C01876=52.817,75.362,62.469,-177.2451,7.5721,0.0000
C01877=50.052,70.729,61.698,-175.7549,6.7538,0.0000
C01878=46.818,66.007,60.151,-176.6982,5.1590,0.0000
C01879=43.998,61.798,58.158,-178.4123,2.6620,0.0000
C01880=42.158,58.431,56.252,178.4711,-3.3109,0.0000
C01881=41.963,55.679,54.888,-171.7704,-29.0710,0.0000
C01882=44.137,52.905,54.350,-151.3798,-29.7512,0.0000
C01883=46.553,50.718,54.326,-149.2273,-28.3546,0.0000
C01884=48.679,48.679,54.342,-150.4011,-29.5986,0.0000
C01885=50.718,46.553,54.326,-151.6456,-30.7729,0.0000
C01886=52.905,44.137,54.350,-150.2477,-28.6184,0.0000
C01887=55.680,41.963,54.888,-150.9289,-8.2300,0.0000
C01888=58.431,42.158,56.252,-176.6891,1.5289,0.0000
C01889=61.798,43.998,58.158,177.3380,-1.5877,0.0000
C01890=66.007,46.818,60.151,174.8410,-3.3018,0.0000
C01891=70.729,50.052,61.698,173.2462,-4.2451,0.0000
C01892=75.362,52.817,62.469,172.4279,-2.7549,0.0000
C01893=80.376,53.158,62.877,175.1551,1.0270,0.0000
C01894=85.074,50.908,63.210,178.0786,1.5643,0.0000
C01895=88.493,46.465,63.547,179.9251,0.1391,0.0000
C01896=91.166,41.080,63.770,179.9921,0.0174,0.0000
C01897=93.512,35.416,63.770,179.9933,0.0179,0.0000
C01898=95.429,29.718,63.547,179.9546,0.1514,0.0000
C01899=96.154,24.159,63.210,-179.7472,2.4641,0.0000
C01900=94.423,19.246,62.877,-177.2942,4.1530,0.0000
C01901=90.636,15.942,62.469,-172.7045,3.4321,0.0000
C01902=85.405,14.621,61.698,-172.2425,1.7901,0.0000
C01903=79.780,13.569,60.151,-174.0266,1.3203,0.0000
C01904=74.809,12.586,58.158,-176.9961,0.7607,0.0000
C01905=71.127,11.507,56.252,176.5790,-1.2623,0.0000
C01906=69.044,9.699,54.888,163.7838,-26.3525,0.0000
C01907=68.619,6.200,54.350,178.9508,-38.3093,0.0000
C01908=68.781,2.945,54.326,-177.7405,-38.7530,0.0000
C01909=68.843,0.000,54.342,-179.9996,-38.7765,0.0000
C01910=68.781,-2.945,54.326,177.7401,-38.7530,0.0000
C01911=68.619,-6.200,54.350,-178.9482,-38.3089,0.0000
C01912=69.044,-9.699,54.888,-163.7840,-26.3528,0.0000
C01913=71.127,-11.507,56.252,-176.5790,-1.2623,0.0000
C01914=74.809,-12.586,58.158,176.9961,0.7607,0.0000
C01915=79.780,-13.569,60.151,174.0266,1.3203,0.0000
C01916=85.405,-14.621,61.698,172.2425,1.7901,0.0000
C01917=90.636,-15.942,62.469,172.7045,3.4321,0.0000
C01918=94.423,-19.246,62.877,177.2942,4.1530,0.0000
C01919=96.154,-24.159,63.210,179.7472,2.4641,0.0000
C01920=95.429,-29.718,63.547,-179.9546,0.1514,0.0000
C01921=93.512,-35.416,63.770,-179.9933,0.0179,0.0000
C01922=91.166,-41.080,63.770,-179.9921,0.0174,0.0000
C01923=88.493,-46.465,63.547,-179.9251,0.1391,0.0000
C01924=85.074,-50.908,63.210,-178.0786,1.5643,0.0000
C01925=80.376,-53.158,62.877,-175.1551,1.0270,0.0000
C01926=75.362,-52.817,62.469,-172.4279,-2.7549,0.0000
C01927=70.729,-50.052,61.698,-173.2462,-4.2451,0.0000
C01928=66.007,-46.818,60.151,-174.8410,-3.3018,0.0000
C01929=61.798,-43.998,58.158,-177.3380,-1.5877,0.0000
C01930=58.431,-42.158,56.252,176.6891,1.5289,0.0000
C01931=55.679,-41.963,54.888,150.9290,-8.2296,0.0000
C01932=52.905,-44.137,54.350,150.2488,-28.6202,0.0000
C01933=50.718,-46.553,54.326,151.6454,-30.7727,0.0000
C01934=48.679,-48.679,54.342,150.4014,-29.5989,0.0000
C01935=46.553,-50.718,54.326,149.2271,-28.3544,0.0000
C01936=44.137,-52.905,54.350,151.3816,-29.7523,0.0000
C01937=41.963,-55.680,54.888,171.7700,-29.0711,0.0000
C01938=42.158,-58.431,56.252,-178.4711,-3.3109,0.0000
C01939=43.998,-61.798,58.158,178.4123,2.6620,0.0000
C01940=46.818,-66.007,60.151,176.6982,5.1590,0.0000
C01941=50.052,-70.729,61.698,175.7549,6.7538,0.0000
C01942=52.817,-75.362,62.469,177.2451,7.5721,0.0000
C01943=53.158,-80.376,62.877,-178.9730,4.8449,0.0000
C01944=50.908,-85.074,63.210,-178.4357,1.9214,0.0000
C01945=46.465,-88.493,63.547,-179.8609,0.0749,0.0000
C01946=41.080,-91.166,63.770,-179.9826,0.0079,0.0000
C01947=35.416,-93.512,63.770,-179.9821,0.0067,0.0000
C01948=29.718,-95.429,63.547,-179.8486,0.0454,0.0000
C01949=24.159,-96.154,63.210,-177.5359,-0.2528,0.0000
C01950=19.246,-94.423,62.877,-175.8470,-2.7058,0.0000
C01951=15.942,-90.636,62.469,-176.5679,-7.2955,0.0000
C01952=14.621,-85.405,61.698,-178.2099,-7.7575,0.0000
C01953=13.569,-79.780,60.151,-178.6797,-5.9734,0.0000
C01954=12.586,-74.809,58.158,-179.2393,-3.0039,0.0000
C01955=11.507,-71.127,56.252,178.7377,3.4210,0.0000
C01956=9.699,-69.044,54.888,153.6475,16.2162,0.0000
C01957=6.200,-68.619,54.350,141.6907,1.0492,0.0000
C01958=2.945,-68.781,54.326,141.2470,-2.2595,0.0000
C01959=0.000,-68.843,54.342,141.2235,-0.0004,0.0000
C01960=0.000,-68.843,54.342,141.2235,-0.0004,0.0000
C01961=-2.945,-68.781,54.326,141.2470,2.2599,0.0000
C01962=-6.200,-68.619,54.350,141.6911,-1.0518,0.0000
C01963=-9.699,-69.044,54.888,153.6472,-16.2160,0.0000
C01964=-11.507,-71.127,56.252,178.7377,-3.4210,0.0000
C01965=-12.586,-74.809,58.158,-179.2393,3.0039,0.0000
C01966=-13.569,-79.780,60.151,-178.6797,5.9734,0.0000
C01967=-14.621,-85.405,61.698,-178.2099,7.7575,0.0000
C01968=-15.942,-90.636,62.469,-176.5679,7.2955,0.0000
C01969=-19.246,-94.423,62.877,-175.8470,2.7058,0.0000
C01970=-24.159,-96.154,63.210,-177.5359,0.2528,0.0000
C01971=-29.718,-95.429,63.547,-179.8486,-0.0454,0.0000
C01972=-35.416,-93.512,63.770,-179.9821,-0.0067,0.0000
C01973=-41.080,-91.166,63.770,-179.9826,-0.0079,0.0000
C01974=-46.465,-88.493,63.547,-179.8609,-0.0749,0.0000
C01975=-50.908,-85.074,63.210,-178.4357,-1.9214,0.0000
C01976=-53.158,-80.376,62.877,-178.9730,-4.8449,0.0000
C01977=-52.817,-75.362,62.469,177.2451,-7.5721,0.0000
C01978=-50.052,-70.729,61.698,175.7549,-6.7538,0.0000
C01979=-46.818,-66.007,60.151,176.6982,-5.1590,0.0000
C01980=-43.998,-61.798,58.158,178.4123,-2.6620,0.0000
C01981=-42.158,-58.431,56.252,-178.4711,3.3109,0.0000
C01982=-41.963,-55.679,54.888,171.7704,29.0710,0.0000
C01983=-44.137,-52.905,54.350,151.3798,29.7512,0.0000
C01984=-46.553,-50.718,54.326,149.2273,28.3546,0.0000
C01985=-48.679,-48.679,54.342,150.4011,29.5986,0.0000
C01986=-50.718,-46.553,54.326,151.6456,30.7729,0.0000
C01987=-52.905,-44.137,54.350,150.2477,28.6184,0.0000
C01988=-55.680,-41.963,54.888,150.9289,8.2300,0.0000
C01989=-58.431,-42.158,56.252,176.6891,-1.5289,0.0000
C01990=-61.798,-43.998,58.158,-177.3380,1.5877,0.0000
C01991=-66.007,-46.818,60.151,-174.8410,3.3018,0.0000
C01992=-70.729,-50.052,61.698,-173.2462,4.2451,0.0000
C01993=-75.362,-52.817,62.469,-172.4279,2.7549,0.0000
C01994=-80.376,-53.158,62.877,-175.1551,-1.0270,0.0000
C01995=-85.074,-50.908,63.210,-178.0786,-1.5643,0.0000
C01996=-88.493,-46.465,63.547,-179.9251,-0.1391,0.0000
C01997=-91.166,-41.080,63.770,-179.9921,-0.0174,0.0000
C01998=-93.512,-35.416,63.770,-179.9933,-0.0179,0.0000
C01999=-95.429,-29.718,63.547,-179.9546,-0.1514,0.0000
///TOOL 0
///POSTYPE ANGLE
///ANGLE
EC00000=-73.7963,0.0000
EC00001=-71.3299,0.0000
EC00002=-68.7820,0.0000
EC00003=-66.2179,0.0000
EC00004=-63.6703,0.0000
EC00005=-61.2039,0.0000
EC00006=-59.0550,0.0000
EC00007=-57.5413,0.0000
EC00008=-56.8513,0.0000
EC00009=-56.3680,0.0000
EC00010=-55.8386,0.0000
EC00011=-55.0278,0.0000
EC00012=-53.5081,0.0000
EC00013=-50.7770,0.0000
EC00014=-47.9180,0.0000
EC00015=-45.0000,0.0000
EC00016=-42.0820,0.0000
EC00017=-39.2230,0.0000
EC00018=-36.4919,0.0000
EC00019=-34.9722,0.0000
EC00020=-34.1614,0.0000
EC00021=-33.6320,0.0000
EC00022=-33.1487,0.0000
EC00023=-32.4587,0.0000
EC00024=-30.9450,0.0000
EC00025=-28.7961,0.0000
EC00026=-26.3297,0.0000
EC00027=-23.7821,0.0000
EC00028=-21.2180,0.0000
EC00029=-18.6701,0.0000
EC00030=-16.2037,0.0000
EC00031=-14.0550,0.0000
EC00032=-12.5410,0.0000
EC00033=-11.8512,0.0000
EC00034=-11.3683,0.0000
EC00035=-10.8382,0.0000
EC00036=-10.0280,0.0000
EC00037=-8.5076,0.0000
EC00038=-5.7775,0.0000
EC00039=-2.9180,0.0000
EC00040=0.0000,0.0000
EC00041=0.0000,0.0000
EC00042=2.8792,0.0000
EC00043=5.7259,0.0000
EC00044=8.4654,0.0000
EC00045=9.9566,0.0000
EC00046=10.7254,0.0000
EC00047=11.2119,0.0000
EC00048=11.6495,0.0000
EC00049=12.2909,0.0000
EC00050=13.8024,0.0000
EC00051=15.9922,0.0000
EC00052=18.5312,0.0000
EC00053=21.1696,0.0000
EC00054=23.8303,0.0000
EC00055=26.4689,0.0000
EC00056=29.0082,0.0000
EC00057=31.1977,0.0000
EC00058=32.7089,0.0000
EC00059=33.3509,0.0000
EC00060=33.7878,0.0000
EC00061=34.2746,0.0000
EC00062=35.0436,0.0000
EC00063=36.5348,0.0000
EC00064=39.2737,0.0000
EC00065=42.1206,0.0000
EC00066=45.0000,0.0000
EC00067=47.8789,0.0000
EC00068=50.7263,0.0000
EC00069=53.4652,0.0000
EC00070=54.9564,0.0000
EC00071=55.7254,0.0000
EC00072=56.2122,0.0000
EC00073=56.6491,0.0000
EC00074=57.2911,0.0000
EC00075=58.8023,0.0000
EC00076=60.9918,0.0000
EC00077=63.5311,0.0000
EC00078=66.1697,0.0000
EC00079=68.8304,0.0000
EC00080=71.4688,0.0000
EC00081=74.0078,0.0000
EC00082=76.1976,0.0000
EC00083=77.7091,0.0000
EC00084=78.3505,0.0000
EC00085=78.7881,0.0000
EC00086=79.2746,0.0000
EC00087=80.0434,0.0000
EC00088=81.5346,0.0000
EC00089=84.2741,0.0000
EC00090=87.1208,0.0000
EC00091=90.0000,0.0000
EC00092=92.8792,0.0000
EC00093=95.7266,0.0000
EC00094=98.4654,0.0000
EC00095=99.9566,0.0000
EC00096=100.7254,0.0000
EC00097=101.2119,0.0000
EC00098=101.6495,0.0000
EC00099=102.2909,0.0000
EC00100=103.8024,0.0000
EC00101=105.9922,0.0000
EC00102=108.5312,0.0000
EC00103=111.1696,0.0000
EC00104=113.8303,0.0000
EC00105=116.4689,0.0000
EC00106=119.0082,0.0000
EC00107=121.1977,0.0000
EC00108=122.7089,0.0000
EC00109=123.3509,0.0000
EC00110=123.7878,0.0000
EC00111=124.2746,0.0000
EC00112=125.0436,0.0000
EC00113=126.5348,0.0000
EC00114=129.2737,0.0000
EC00115=132.1206,0.0000
EC00116=135.0000,0.0000
EC00117=137.8789,0.0000
EC00118=140.7263,0.0000
EC00119=143.4652,0.0000
EC00120=144.9564,0.0000
EC00121=145.7254,0.0000
EC00122=146.2122,0.0000
EC00123=146.6491,0.0000
EC00124=147.2911,0.0000
EC00125=148.8023,0.0000
EC00126=150.9918,0.0000
EC00127=153.5311,0.0000
EC00128=156.1697,0.0000
EC00129=158.8304,0.0000
EC00130=161.4688,0.0000
EC00131=164.0078,0.0000
EC00132=166.1976,0.0000
EC00133=167.7091,0.0000
EC00134=168.3505,0.0000
EC00135=168.7881,0.0000
EC00136=169.2746,0.0000
EC00137=170.0434,0.0000
EC00138=171.5346,0.0000
EC00139=174.2741,0.0000
EC00140=177.1208,0.0000
EC00141=180.0000,0.0000
EC00142=180.0000,0.0000
EC00143=-177.1208,0.0000
EC00144=-174.2734,0.0000
EC00145=-171.5346,0.0000
EC00146=-170.0434,0.0000
EC00147=-169.2746,0.0000
EC00148=-168.7881,0.0000
EC00149=-168.3505,0.0000
EC00150=-167.7091,0.0000
EC00151=-166.1976,0.0000
EC00152=-164.0078,0.0000
EC00153=-161.4688,0.0000
EC00154=-158.8304,0.0000
EC00155=-156.1697,0.0000
EC00156=-153.5311,0.0000
EC00157=-150.9918,0.0000
EC00158=-148.8023,0.0000
EC00159=-147.2911,0.0000
EC00160=-146.6491,0.0000
EC00161=-146.2122,0.0000
EC00162=-145.7254,0.0000
EC00163=-144.9564,0.0000
EC00164=-143.4652,0.0000
EC00165=-140.7263,0.0000
EC00166=-137.8794,0.0000
EC00167=-135.0000,0.0000
EC00168=-132.1211,0.0000
EC00169=-129.2737,0.0000
EC00170=-126.5348,0.0000
EC00171=-125.0436,0.0000
EC00172=-124.2746,0.0000
EC00173=-123.7878,0.0000
EC00174=-123.3509,0.0000
EC00175=-122.7089,0.0000
EC00176=-121.1977,0.0000
EC00177=-119.0082,0.0000
EC00178=-116.4689,0.0000
EC00179=-113.8303,0.0000
EC00180=-111.1696,0.0000
EC00181=-108.5312,0.0000
EC00182=-105.9922,0.0000
EC00183=-103.8024,0.0000
EC00184=-102.2909,0.0000
EC00185=-101.6495,0.0000
EC00186=-101.2119,0.0000
EC00187=-100.7254,0.0000
EC00188=-99.9566,0.0000
EC00189=-98.4654,0.0000
EC00190=-95.7259,0.0000
EC00191=-92.8792,0.0000
EC00192=-90.0000,0.0000
EC00193=-87.1208,0.0000
EC00194=-84.2734,0.0000
EC00195=-81.5346,0.0000
EC00196=-80.0434,0.0000
EC00197=-79.2746,0.0000
EC00198=-78.7881,0.0000
EC00199=-78.3505,0.0000
EC00200=-77.7091,0.0000
EC00201=-76.1976,0.0000
EC00202=-74.0078,0.0000
EC00203=-71.4688,0.0000
EC00204=-68.8304,0.0000
EC00205=-66.1697,0.0000
EC00206=-63.5311,0.0000
EC00207=-60.9918,0.0000
EC00208=-58.8023,0.0000
EC00209=-57.2911,0.0000
EC00210=-56.6491,0.0000
EC00211=-56.2122,0.0000
EC00212=-55.7254,0.0000
EC00213=-54.9564,0.0000
EC00214=-53.4652,0.0000
EC00215=-50.7263,0.0000
EC00216=-47.8794,0.0000
EC00217=-45.0000,0.0000
EC00218=-42.1211,0.0000
EC00219=-39.2737,0.0000
EC00220=-36.5348,0.0000
EC00221=-35.0436,0.0000
EC00222=-34.2746,0.0000
EC00223=-33.7878,0.0000
EC00224=-33.3509,0.0000
EC00225=-32.7089,0.0000
EC00226=-31.1977,0.0000
EC00227=-29.0082,0.0000
EC00228=-26.4689,0.0000
EC00229=-23.8303,0.0000
EC00230=-21.1696,0.0000
EC00231=-18.5312,0.0000
EC00232=-15.9922,0.0000
EC00233=-13.8024,0.0000
EC00234=-12.2909,0.0000
EC00235=-11.6495,0.0000
EC00236=-11.2119,0.0000
EC00237=-10.7254,0.0000
EC00238=-9.9566,0.0000
EC00239=-8.4654,0.0000
EC00240=-5.7266,0.0000
EC00241=-2.8792,0.0000
EC00242=0.0000,0.0000
EC00243=0.0000,0.0000
EC00244=2.8388,0.0000
EC00245=5.6728,0.0000
EC00246=8.4202,0.0000
EC00247=9.8823,0.0000
EC00248=10.6084,0.0000
EC00249=11.0516,0.0000
EC00250=11.4429,0.0000
EC00251=12.0370,0.0000
EC00252=13.5473,0.0000
EC00253=15.7781,0.0000
EC00254=18.3907,0.0000
EC00255=21.1209,0.0000
EC00256=23.8793,0.0000
EC00257=26.6097,0.0000
EC00258=29.2218,0.0000
EC00259=31.4529,0.0000
EC00260=32.9628,0.0000
EC00261=33.5569,0.0000
EC00262=33.9481,0.0000
EC00263=34.3909,0.0000
EC00264=35.1173,0.0000
EC00265=36.5793,0.0000
EC00266=39.3269,0.0000
EC00267=42.1606,0.0000
EC00268=45.0000,0.0000
EC00269=47.8388,0.0000
EC00270=50.6731,0.0000
EC00271=53.4207,0.0000
EC00272=54.8827,0.0000
EC00273=55.6091,0.0000
EC00274=56.0519,0.0000
EC00275=56.4431,0.0000
EC00276=57.0372,0.0000
EC00277=58.5471,0.0000
EC00278=60.7782,0.0000
EC00279=63.3903,0.0000
EC00280=66.1207,0.0000
EC00281=68.8791,0.0000
EC00282=71.6093,0.0000
EC00283=74.2219,0.0000
EC00284=76.4527,0.0000
EC00285=77.9630,0.0000
EC00286=78.5571,0.0000
EC00287=78.9484,0.0000
EC00288=79.3916,0.0000
EC00289=80.1177,0.0000
EC00290=81.5798,0.0000
EC00291=84.3272,0.0000
EC00292=87.1612,0.0000
EC00293=90.0000,0.0000
EC00294=92.8388,0.0000
EC00295=95.6728,0.0000
EC00296=98.4209,0.0000
EC00297=99.8823,0.0000
EC00298=100.6084,0.0000
EC00299=101.0516,0.0000
EC00300=101.4429,0.0000
EC00301=102.0370,0.0000
EC00302=103.5473,0.0000
EC00303=105.7781,0.0000
EC00304=108.3907,0.0000
EC00305=111.1209,0.0000
EC00306=113.8793,0.0000
EC00307=116.6097,0.0000
EC00308=119.2218,0.0000
EC00309=121.4529,0.0000
EC00310=122.9628,0.0000
EC00311=123.5569,0.0000
EC00312=123.9481,0.0000
EC00313=124.3909,0.0000
EC00314=125.1173,0.0000
EC00315=126.5793,0.0000
EC00316=129.3269,0.0000
EC00317=132.1606,0.0000
EC00318=135.0000,0.0000
EC00319=137.8388,0.0000
EC00320=140.6731,0.0000
EC00321=143.4207,0.0000
EC00322=144.8827,0.0000
EC00323=145.6091,0.0000
EC00324=146.0519,0.0000
EC00325=146.4431,0.0000
EC00326=147.0372,0.0000
EC00327=148.5471,0.0000
EC00328=150.7782,0.0000
EC00329=153.3903,0.0000
EC00330=156.1207,0.0000
EC00331=158.8791,0.0000
EC00332=161.6093,0.0000
EC00333=164.2219,0.0000
EC00334=166.4527,0.0000
EC00335=167.9630,0.0000
EC00336=168.5571,0.0000
EC00337=168.9484,0.0000
EC00338=169.3916,0.0000
EC00339=170.1177,0.0000
EC00340=171.5798,0.0000
EC00341=174.3272,0.0000
EC00342=177.1612,0.0000
EC00343=180.0000,0.0000
EC00344=180.0000,0.0000
EC00345=-177.1612,0.0000
EC00346=-174.3272,0.0000
EC00347=-171.5791,0.0000
EC00348=-170.1177,0.0000
EC00349=-169.3916,0.0000
EC00350=-168.9484,0.0000
EC00351=-168.5571,0.0000
EC00352=-167.9630,0.0000
EC00353=-166.4527,0.0000
EC00354=-164.2219,0.0000
EC00355=-161.6093,0.0000
EC00356=-158.8791,0.0000
EC00357=-156.1207,0.0000
EC00358=-153.3903,0.0000
EC00359=-150.7782,0.0000
EC00360=-148.5471,0.0000
EC00361=-147.0372,0.0000
EC00362=-146.4431,0.0000
EC00363=-146.0519,0.0000
EC00364=-145.6091,0.0000
EC00365=-144.8827,0.0000
EC00366=-143.4207,0.0000
EC00367=-140.6731,0.0000
EC00368=-137.8394,0.0000
EC00369=-135.0000,0.0000
EC00370=-132.1612,0.0000
EC00371=-129.3269,0.0000
EC00372=-126.5793,0.0000
EC00373=-125.1173,0.0000
EC00374=-124.3909,0.0000
EC00375=-123.9481,0.0000
EC00376=-123.5569,0.0000
EC00377=-122.9628,0.0000
EC00378=-121.4529,0.0000
EC00379=-119.2218,0.0000
EC00380=-116.6097,0.0000
EC00381=-113.8793,0.0000
EC00382=-111.1209,0.0000
EC00383=-108.3907,0.0000
EC00384=-105.7781,0.0000
EC00385=-103.5473,0.0000
EC00386=-102.0370,0.0000
EC00387=-101.4429,0.0000
EC00388=-101.0516,0.0000
EC00389=-100.6084,0.0000
EC00390=-99.8823,0.0000
EC00391=-98.4202,0.0000
EC00392=-95.6728,0.0000
EC00393=-92.8388,0.0000
EC00394=-90.0000,0.0000
EC00395=-87.1612,0.0000
EC00396=-84.3272,0.0000
EC00397=-81.5791,0.0000
EC00398=-80.1177,0.0000
EC00399=-79.3916,0.0000
EC00400=-78.9484,0.0000
EC00401=-78.5571,0.0000
EC00402=-77.9630,0.0000
EC00403=-76.4527,0.0000
EC00404=-74.2219,0.0000
EC00405=-71.6093,0.0000
EC00406=-68.8791,0.0000
EC00407=-66.1207,0.0000
EC00408=-63.3903,0.0000
EC00409=-60.7782,0.0000
EC00410=-58.5471,0.0000
EC00411=-57.0372,0.0000
EC00412=-56.4431,0.0000
EC00413=-56.0519,0.0000
EC00414=-55.6091,0.0000
EC00415=-54.8827,0.0000
EC00416=-53.4207,0.0000
EC00417=-50.6731,0.0000
EC00418=-47.8394,0.0000
EC00419=-45.0000,0.0000
EC00420=-42.1612,0.0000
EC00421=-39.3269,0.0000
EC00422=-36.5793,0.0000
EC00423=-35.1173,0.0000
EC00424=-34.3909,0.0000
EC00425=-33.9481,0.0000
EC00426=-33.5569,0.0000
EC00427=-32.9628,0.0000
EC00428=-31.4529,0.0000
EC00429=-29.2218,0.0000
EC00430=-26.6097,0.0000
EC00431=-23.8793,0.0000
EC00432=-21.1209,0.0000
EC00433=-18.3907,0.0000
EC00434=-15.7781,0.0000
EC00435=-13.5473,0.0000
EC00436=-12.0370,0.0000
EC00437=-11.4429,0.0000
EC00438=-11.0516,0.0000
EC00439=-10.6084,0.0000
EC00440=-9.8823,0.0000
EC00441=-8.4209,0.0000
EC00442=-5.6728,0.0000
EC00443=-2.8388,0.0000
EC00444=0.0000,0.0000
EC00445=0.0000,0.0000
EC00446=2.7966,0.0000
EC00447=5.6177,0.0000
EC00448=8.3745,0.0000
EC00449=9.8055,0.0000
EC00450=10.4884,0.0000
EC00451=10.8872,0.0000
EC00452=11.2331,0.0000
EC00453=11.7800,0.0000
EC00454=13.2896,0.0000
EC00455=15.5634,0.0000
EC00456=18.2498,0.0000
EC00457=21.0723,0.0000
EC00458=23.9275,0.0000
EC00459=26.7502,0.0000
EC00460=29.4368,0.0000
EC00461=31.7100,0.0000
EC00462=33.2198,0.0000
EC00463=33.7669,0.0000
EC00464=34.1127,0.0000
EC00465=34.5119,0.0000
EC00466=35.1948,0.0000
EC00467=36.6259,0.0000
EC00468=39.3828,0.0000
EC00469=42.2032,0.0000
EC00470=45.0000,0.0000
EC00471=47.7968,0.0000
EC00472=50.6172,0.0000
EC00473=53.3741,0.0000
EC00474=54.8052,0.0000
EC00475=55.4881,0.0000
EC00476=55.8873,0.0000
EC00477=56.2331,0.0000
EC00478=56.7802,0.0000
EC00479=58.2900,0.0000
EC00480=60.5632,0.0000
EC00481=63.2498,0.0000
EC00482=66.0725,0.0000
EC00483=68.9277,0.0000
EC00484=71.7502,0.0000
EC00485=74.4366,0.0000
EC00486=76.7104,0.0000
EC00487=78.2200,0.0000
EC00488=78.7669,0.0000
EC00489=79.1128,0.0000
EC00490=79.5116,0.0000
EC00491=80.1945,0.0000
EC00492=81.6255,0.0000
EC00493=84.3823,0.0000
EC00494=87.2034,0.0000
EC00495=90.0000,0.0000
EC00496=92.7966,0.0000
EC00497=95.6177,0.0000
EC00498=98.3745,0.0000
EC00499=99.8055,0.0000
EC00500=100.4884,0.0000
EC00501=100.8872,0.0000
EC00502=101.2331,0.0000
EC00503=101.7800,0.0000
EC00504=103.2896,0.0000
EC00505=105.5634,0.0000
EC00506=108.2498,0.0000
EC00507=111.0723,0.0000
EC00508=113.9275,0.0000
EC00509=116.7502,0.0000
EC00510=119.4368,0.0000
EC00511=121.7100,0.0000
EC00512=123.2198,0.0000
EC00513=123.7669,0.0000
EC00514=124.1127,0.0000
EC00515=124.5119,0.0000
EC00516=125.1948,0.0000
EC00517=126.6259,0.0000
EC00518=129.3828,0.0000
EC00519=132.2032,0.0000
EC00520=135.0000,0.0000
EC00521=137.7968,0.0000
EC00522=140.6172,0.0000
EC00523=143.3741,0.0000
EC00524=144.8052,0.0000
EC00525=145.4881,0.0000
EC00526=145.8873,0.0000
EC00527=146.2331,0.0000
EC00528=146.7802,0.0000
EC00529=148.2900,0.0000
EC00530=150.5632,0.0000
EC00531=153.2498,0.0000
EC00532=156.0725,0.0000
EC00533=158.9277,0.0000
EC00534=161.7502,0.0000
EC00535=164.4366,0.0000
EC00536=166.7104,0.0000
EC00537=168.2200,0.0000
EC00538=168.7669,0.0000
EC00539=169.1128,0.0000
EC00540=169.5116,0.0000
EC00541=170.1945,0.0000
EC00542=171.6255,0.0000
EC00543=174.3823,0.0000
EC00544=177.2034,0.0000
EC00545=180.0000,0.0000
EC00546=180.0000,0.0000
EC00547=-177.2034,0.0000
EC00548=-174.3823,0.0000
EC00549=-171.6255,0.0000
EC00550=-170.1945,0.0000
EC00551=-169.5116,0.0000
EC00552=-169.1128,0.0000
EC00553=-168.7669,0.0000
EC00554=-168.2200,0.0000
EC00555=-166.7104,0.0000
EC00556=-164.4366,0.0000
EC00557=-161.7502,0.0000
EC00558=-158.9277,0.0000
EC00559=-156.0725,0.0000
EC00560=-153.2498,0.0000
EC00561=-150.5632,0.0000
EC00562=-148.2900,0.0000
EC00563=-146.7802,0.0000
EC00564=-146.2331,0.0000
EC00565=-145.8873,0.0000
EC00566=-145.4881,0.0000
EC00567=-144.8052,0.0000
EC00568=-143.3741,0.0000
EC00569=-140.6172,0.0000
EC00570=-137.7968,0.0000
EC00571=-135.0000,0.0000
EC00572=-132.2032,0.0000
EC00573=-129.3828,0.0000
EC00574=-126.6259,0.0000
EC00575=-125.1948,0.0000
EC00576=-124.5119,0.0000
EC00577=-124.1127,0.0000
EC00578=-123.7669,0.0000
EC00579=-123.2198,0.0000
EC00580=-121.7100,0.0000
EC00581=-119.4368,0.0000
EC00582=-116.7502,0.0000
EC00583=-113.9275,0.0000
EC00584=-111.0723,0.0000
EC00585=-108.2498,0.0000
EC00586=-105.5634,0.0000
EC00587=-103.2896,0.0000
EC00588=-101.7800,0.0000
EC00589=-101.2331,0.0000
EC00590=-100.8872,0.0000
EC00591=-100.4884,0.0000
EC00592=-99.8055,0.0000
EC00593=-98.3745,0.0000
EC00594=-95.6177,0.0000
EC00595=-92.7966,0.0000
EC00596=-90.0000,0.0000
EC00597=-87.2034,0.0000
EC00598=-84.3823,0.0000
EC00599=-81.6255,0.0000
EC00600=-80.1945,0.0000
EC00601=-79.5116,0.0000
EC00602=-79.1128,0.0000
EC00603=-78.7669,0.0000
EC00604=-78.2200,0.0000
EC00605=-76.7104,0.0000
EC00606=-74.4366,0.0000
EC00607=-71.7502,0.0000
EC00608=-68.9277,0.0000
EC00609=-66.0725,0.0000
EC00610=-63.2498,0.0000
EC00611=-60.5632,0.0000
EC00612=-58.2900,0.0000
EC00613=-56.7802,0.0000
EC00614=-56.2331,0.0000
EC00615=-55.8873,0.0000
EC00616=-55.4881,0.0000
EC00617=-54.8052,0.0000
EC00618=-53.3741,0.0000
EC00619=-50.6172,0.0000
EC00620=-47.7968,0.0000
EC00621=-45.0000,0.0000
EC00622=-42.2032,0.0000
EC00623=-39.3828,0.0000
EC00624=-36.6259,0.0000
EC00625=-35.1948,0.0000
EC00626=-34.5119,0.0000
EC00627=-34.1127,0.0000
EC00628=-33.7669,0.0000
EC00629=-33.2198,0.0000
EC00630=-31.7100,0.0000
EC00631=-29.4368,0.0000
EC00632=-26.7502,0.0000
EC00633=-23.9275,0.0000
EC00634=-21.0723,0.0000
EC00635=-18.2498,0.0000
EC00636=-15.5634,0.0000
EC00637=-13.2896,0.0000
EC00638=-11.7800,0.0000
EC00639=-11.2331,0.0000
EC00640=-10.8872,0.0000
EC00641=-10.4884,0.0000
EC00642=-9.8055,0.0000
EC00643=-8.3745,0.0000
EC00644=-5.6177,0.0000
EC00645=-2.7966,0.0000
EC00646=0.0000,0.0000
EC00647=0.0000,0.0000
EC00648=2.7531,0.0000
EC00649=5.5598,0.0000
EC00650=8.3257,0.0000
EC00651=9.7254,0.0000
EC00652=10.3637,0.0000
EC00653=10.7187,0.0000
EC00654=11.0200,0.0000
EC00655=11.5211,0.0000
EC00656=13.0317,0.0000
EC00657=15.3479,0.0000
EC00658=18.1086,0.0000
EC00659=21.0234,0.0000
EC00660=23.9765,0.0000
EC00661=26.8914,0.0000
EC00662=29.6519,0.0000
EC00663=31.9680,0.0000
EC00664=33.4791,0.0000
EC00665=33.9803,0.0000
EC00666=34.2813,0.0000
EC00667=34.6359,0.0000
EC00668=35.2745,0.0000
EC00669=36.6744,0.0000
EC00670=39.4401,0.0000
EC00671=42.2471,0.0000
EC00672=45.0000,0.0000
EC00673=47.7529,0.0000
EC00674=50.5599,0.0000
EC00675=53.3256,0.0000
EC00676=54.7255,0.0000
EC00677=55.3641,0.0000
EC00678=55.7187,0.0000
EC00679=56.0197,0.0000
EC00680=56.5209,0.0000
EC00681=58.0320,0.0000
EC00682=60.3481,0.0000
EC00683=63.1086,0.0000
EC00684=66.0235,0.0000
EC00685=68.9766,0.0000
EC00686=71.8914,0.0000
EC00687=74.6521,0.0000
EC00688=76.9683,0.0000
EC00689=78.4789,0.0000
EC00690=78.9800,0.0000
EC00691=79.2813,0.0000
EC00692=79.6363,0.0000
EC00693=80.2746,0.0000
EC00694=81.6743,0.0000
EC00695=84.4402,0.0000
EC00696=87.2469,0.0000
EC00697=90.0000,0.0000
EC00698=92.7531,0.0000
EC00699=95.5598,0.0000
EC00700=98.3257,0.0000
EC00701=99.7254,0.0000
EC00702=100.3637,0.0000
EC00703=100.7187,0.0000
EC00704=101.0200,0.0000
EC00705=101.5211,0.0000
EC00706=103.0317,0.0000
EC00707=105.3479,0.0000
EC00708=108.1086,0.0000
EC00709=111.0234,0.0000
EC00710=113.9765,0.0000
EC00711=116.8914,0.0000
EC00712=119.6519,0.0000
EC00713=121.9680,0.0000
EC00714=123.4791,0.0000
EC00715=123.9803,0.0000
EC00716=124.2813,0.0000
EC00717=124.6359,0.0000
EC00718=125.2745,0.0000
EC00719=126.6744,0.0000
EC00720=129.4401,0.0000
EC00721=132.2471,0.0000
EC00722=135.0000,0.0000
EC00723=137.7529,0.0000
EC00724=140.5599,0.0000
EC00725=143.3256,0.0000
EC00726=144.7255,0.0000
EC00727=145.3641,0.0000
EC00728=145.7187,0.0000
EC00729=146.0197,0.0000
EC00730=146.5209,0.0000
EC00731=148.0320,0.0000
EC00732=150.3481,0.0000
EC00733=153.1086,0.0000
EC00734=156.0235,0.0000
EC00735=158.9766,0.0000
EC00736=161.8914,0.0000
EC00737=164.6521,0.0000
EC00738=166.9683,0.0000
EC00739=168.4789,0.0000
EC00740=168.9800,0.0000
EC00741=169.2813,0.0000
EC00742=169.6363,0.0000
EC00743=170.2746,0.0000
EC00744=171.6743,0.0000
EC00745=174.4402,0.0000
EC00746=177.2469,0.0000
EC00747=180.0000,0.0000
EC00748=180.0000,0.0000
EC00749=-177.2469,0.0000
EC00750=-174.4402,0.0000
EC00751=-171.6743,0.0000
EC00752=-170.2746,0.0000
EC00753=-169.6363,0.0000
EC00754=-169.2813,0.0000
EC00755=-168.9800,0.0000
EC00756=-168.4789,0.0000
EC00757=-166.9683,0.0000
EC00758=-164.6521,0.0000
EC00759=-161.8914,0.0000
EC00760=-158.9766,0.0000
EC00761=-156.0235,0.0000
EC00762=-153.1086,0.0000
EC00763=-150.3481,0.0000
EC00764=-148.0320,0.0000
EC00765=-146.5209,0.0000
EC00766=-146.0197,0.0000
EC00767=-145.7187,0.0000
EC00768=-145.3641,0.0000
EC00769=-144.7255,0.0000
EC00770=-143.3256,0.0000
EC00771=-140.5599,0.0000
EC00772=-137.7529,0.0000
EC00773=-135.0000,0.0000
EC00774=-132.2471,0.0000
EC00775=-129.4401,0.0000
EC00776=-126.6744,0.0000
EC00777=-125.2745,0.0000
EC00778=-124.6359,0.0000
EC00779=-124.2813,0.0000
EC00780=-123.9803,0.0000
EC00781=-123.4791,0.0000
EC00782=-121.9680,0.0000
EC00783=-119.6519,0.0000
EC00784=-116.8914,0.0000
EC00785=-113.9765,0.0000
EC00786=-111.0234,0.0000
EC00787=-108.1086,0.0000
EC00788=-105.3479,0.0000
EC00789=-103.0317,0.0000
EC00790=-101.5211,0.0000
EC00791=-101.0200,0.0000
EC00792=-100.7187,0.0000
EC00793=-100.3637,0.0000
EC00794=-99.7254,0.0000
EC00795=-98.3257,0.0000
EC00796=-95.5598,0.0000
EC00797=-92.7531,0.0000
EC00798=-90.0000,0.0000
EC00799=-87.2469,0.0000
EC00800=-84.4402,0.0000
EC00801=-81.6743,0.0000
EC00802=-80.2746,0.0000
EC00803=-79.6363,0.0000
EC00804=-79.2813,0.0000
EC00805=-78.9800,0.0000
EC00806=-78.4789,0.0000
EC00807=-76.9683,0.0000
EC00808=-74.6521,0.0000
EC00809=-71.8914,0.0000
EC00810=-68.9766,0.0000
EC00811=-66.0235,0.0000
EC00812=-63.1086,0.0000
EC00813=-60.3481,0.0000
EC00814=-58.0320,0.0000
EC00815=-56.5209,0.0000
EC00816=-56.0197,0.0000
EC00817=-55.7187,0.0000
EC00818=-55.3641,0.0000
EC00819=-54.7255,0.0000
EC00820=-53.3256,0.0000
EC00821=-50.5599,0.0000
EC00822=-47.7529,0.0000
EC00823=-45.0000,0.0000
EC00824=-42.2471,0.0000
EC00825=-39.4401,0.0000
EC00826=-36.6744,0.0000
EC00827=-35.2745,0.0000
EC00828=-34.6359,0.0000
EC00829=-34.2813,0.0000
EC00830=-33.9803,0.0000
EC00831=-33.4791,0.0000
EC00832=-31.9680,0.0000
EC00833=-29.6519,0.0000
EC00834=-26.8914,0.0000
EC00835=-23.9765,0.0000
EC00836=-21.0234,0.0000
EC00837=-18.1086,0.0000
EC00838=-15.3479,0.0000
EC00839=-13.0317,0.0000
EC00840=-11.5211,0.0000
EC00841=-11.0200,0.0000
EC00842=-10.7187,0.0000
EC00843=-10.3637,0.0000
EC00844=-9.7254,0.0000
EC00845=-8.3257,0.0000
EC00846=-5.5598,0.0000
EC00847=-2.7531,0.0000
EC00848=0.0000,0.0000
EC00849=0.0000,0.0000
EC00850=2.7075,0.0000
EC00851=5.4993,0.0000
EC00852=8.2758,0.0000
EC00853=9.6431,0.0000
EC00854=10.2359,0.0000
EC00855=10.5465,0.0000
EC00856=10.8039,0.0000
EC00857=11.2607,0.0000
EC00858=12.7735,0.0000
EC00859=15.1340,0.0000
EC00860=17.9686,0.0000
EC00861=20.9753,0.0000
EC00862=24.0247,0.0000
EC00863=27.0314,0.0000
EC00864=29.8659,0.0000
EC00865=32.2261,0.0000
EC00866=33.7397,0.0000
EC00867=34.1962,0.0000
EC00868=34.4534,0.0000
EC00869=34.7640,0.0000
EC00870=35.3567,0.0000
EC00871=36.7241,0.0000
EC00872=39.5007,0.0000
EC00873=42.2930,0.0000
EC00874=45.0000,0.0000
EC00875=47.7070,0.0000
EC00876=50.4999,0.0000
EC00877=53.2759,0.0000
EC00878=54.6433,0.0000
EC00879=55.2360,0.0000
EC00880=55.5466,0.0000
EC00881=55.8038,0.0000
EC00882=56.2603,0.0000
EC00883=57.7739,0.0000
EC00884=60.1341,0.0000
EC00885=62.9686,0.0000
EC00886=65.9753,0.0000
EC00887=69.0247,0.0000
EC00888=72.0314,0.0000
EC00889=74.8660,0.0000
EC00890=77.2265,0.0000
EC00891=78.7393,0.0000
EC00892=79.1961,0.0000
EC00893=79.4535,0.0000
EC00894=79.7641,0.0000
EC00895=80.3569,0.0000
EC00896=81.7242,0.0000
EC00897=84.5007,0.0000
EC00898=87.2925,0.0000
EC00899=90.0000,0.0000
EC00900=92.7075,0.0000
EC00901=95.4993,0.0000
EC00902=98.2758,0.0000
EC00903=99.6431,0.0000
EC00904=100.2359,0.0000
EC00905=100.5465,0.0000
EC00906=100.8039,0.0000
EC00907=101.2607,0.0000
EC00908=102.7735,0.0000
EC00909=105.1340,0.0000
EC00910=107.9686,0.0000
EC00911=110.9753,0.0000
EC00912=114.0247,0.0000
EC00913=117.0314,0.0000
EC00914=119.8659,0.0000
EC00915=122.2261,0.0000
EC00916=123.7397,0.0000
EC00917=124.1962,0.0000
EC00918=124.4534,0.0000
EC00919=124.7640,0.0000
EC00920=125.3567,0.0000
EC00921=126.7241,0.0000
EC00922=129.5007,0.0000
EC00923=132.2930,0.0000
EC00924=135.0000,0.0000
EC00925=137.7070,0.0000
EC00926=140.4999,0.0000
EC00927=143.2759,0.0000
EC00928=144.6433,0.0000
EC00929=145.2360,0.0000
EC00930=145.5466,0.0000
EC00931=145.8038,0.0000
EC00932=146.2603,0.0000
EC00933=147.7739,0.0000
EC00934=150.1341,0.0000
EC00935=152.9686,0.0000
EC00936=155.9753,0.0000
EC00937=159.0247,0.0000
EC00938=162.0314,0.0000
EC00939=164.8660,0.0000
EC00940=167.2265,0.0000
EC00941=168.7393,0.0000
EC00942=169.1961,0.0000
EC00943=169.4535,0.0000
EC00944=169.7641,0.0000
EC00945=170.3569,0.0000
EC00946=171.7242,0.0000
EC00947=174.5007,0.0000
EC00948=177.2925,0.0000
EC00949=180.0000,0.0000
EC00950=180.0000,0.0000
EC00951=-177.2925,0.0000
EC00952=-174.5007,0.0000
EC00953=-171.7242,0.0000
EC00954=-170.3569,0.0000
EC00955=-169.7641,0.0000
EC00956=-169.4535,0.0000
EC00957=-169.1961,0.0000
EC00958=-168.7393,0.0000
EC00959=-167.2265,0.0000
EC00960=-164.8660,0.0000
EC00961=-162.0314,0.0000
EC00962=-159.0247,0.0000
EC00963=-155.9753,0.0000
EC00964=-152.9686,0.0000
EC00965=-150.1341,0.0000
EC00966=-147.7739,0.0000
EC00967=-146.2603,0.0000
EC00968=-145.8038,0.0000
EC00969=-145.5466,0.0000
EC00970=-145.2360,0.0000
EC00971=-144.6433,0.0000
EC00972=-143.2759,0.0000
EC00973=-140.4993,0.0000
EC00974=-137.7070,0.0000
EC00975=-135.0000,0.0000
EC00976=-132.2930,0.0000
EC00977=-129.5001,0.0000
EC00978=-126.7241,0.0000
EC00979=-125.3567,0.0000
EC00980=-124.7640,0.0000
EC00981=-124.4534,0.0000
EC00982=-124.1962,0.0000
EC00983=-123.7397,0.0000
EC00984=-122.2261,0.0000
EC00985=-119.8659,0.0000
EC00986=-117.0314,0.0000
EC00987=-114.0247,0.0000
EC00988=-110.9753,0.0000
EC00989=-107.9686,0.0000
EC00990=-105.1340,0.0000
EC00991=-102.7735,0.0000
EC00992=-101.2607,0.0000
EC00993=-100.8039,0.0000
EC00994=-100.5465,0.0000
EC00995=-100.2359,0.0000
EC00996=-99.6431,0.0000
EC00997=-98.2758,0.0000
EC00998=-95.4993,0.0000
EC00999=-92.7075,0.0000
EC01000=-90.0000,0.0000
EC01001=-87.2925,0.0000
EC01002=-84.5007,0.0000
EC01003=-81.7242,0.0000
EC01004=-80.3569,0.0000
EC01005=-79.7641,0.0000
EC01006=-79.4535,0.0000
EC01007=-79.1961,0.0000
EC01008=-78.7393,0.0000
EC01009=-77.2265,0.0000
EC01010=-74.8660,0.0000
EC01011=-72.0314,0.0000
EC01012=-69.0247,0.0000
EC01013=-65.9753,0.0000
EC01014=-62.9686,0.0000
EC01015=-60.1341,0.0000
EC01016=-57.7739,0.0000
EC01017=-56.2603,0.0000
EC01018=-55.8038,0.0000
EC01019=-55.5466,0.0000
EC01020=-55.2360,0.0000
EC01021=-54.6433,0.0000
EC01022=-53.2759,0.0000
EC01023=-50.4993,0.0000
EC01024=-47.7070,0.0000
EC01025=-45.0000,0.0000
EC01026=-42.2930,0.0000
EC01027=-39.5001,0.0000
EC01028=-36.7241,0.0000
EC01029=-35.3567,0.0000
EC01030=-34.7640,0.0000
EC01031=-34.4534,0.0000
EC01032=-34.1962,0.0000
EC01033=-33.7397,0.0000
EC01034=-32.2261,0.0000
EC01035=-29.8659,0.0000
EC01036=-27.0314,0.0000
EC01037=-24.0247,0.0000
EC01038=-20.9753,0.0000
EC01039=-17.9686,0.0000
EC01040=-15.1340,0.0000
EC01041=-12.7735,0.0000
EC01042=-11.2607,0.0000
EC01043=-10.8039,0.0000
EC01044=-10.5465,0.0000
EC01045=-10.2359,0.0000
EC01046=-9.6431,0.0000
EC01047=-8.2758,0.0000
EC01048=-5.4993,0.0000
EC01049=-2.7075,0.0000
EC01050=0.0000,0.0000
EC01051=0.0000,0.0000
EC01052=2.6603,0.0000
EC01053=5.4368,0.0000
EC01054=8.2235,0.0000
EC01055=9.5577,0.0000
EC01056=10.1045,0.0000
EC01057=10.3719,0.0000
EC01058=10.5864,0.0000
EC01059=10.9998,0.0000
EC01060=12.5167,0.0000
EC01061=14.9212,0.0000
EC01062=17.8298,0.0000
EC01063=20.9268,0.0000
EC01064=24.0730,0.0000
EC01065=27.1707,0.0000
EC01066=30.0788,0.0000
EC01067=32.4830,0.0000
EC01068=34.0000,0.0000
EC01069=34.4140,0.0000
EC01070=34.6279,0.0000
EC01071=34.8952,0.0000
EC01072=35.4421,0.0000
EC01073=36.7764,0.0000
EC01074=39.5628,0.0000
EC01075=42.3404,0.0000
EC01076=45.0000,0.0000
EC01077=47.6596,0.0000
EC01078=50.4372,0.0000
EC01079=53.2236,0.0000
EC01080=54.5579,0.0000
EC01081=55.1048,0.0000
EC01082=55.3721,0.0000
EC01083=55.5860,0.0000
EC01084=56.0000,0.0000
EC01085=57.5170,0.0000
EC01086=59.9212,0.0000
EC01087=62.8293,0.0000
EC01088=65.9270,0.0000
EC01089=69.0732,0.0000
EC01090=72.1702,0.0000
EC01091=75.0788,0.0000
EC01092=77.4833,0.0000
EC01093=79.0002,0.0000
EC01094=79.4136,0.0000
EC01095=79.6281,0.0000
EC01096=79.8955,0.0000
EC01097=80.4423,0.0000
EC01098=81.7765,0.0000
EC01099=84.5632,0.0000
EC01100=87.3397,0.0000
EC01101=90.0000,0.0000
EC01102=92.6603,0.0000
EC01103=95.4368,0.0000
EC01104=98.2235,0.0000
EC01105=99.5577,0.0000
EC01106=100.1045,0.0000
EC01107=100.3719,0.0000
EC01108=100.5864,0.0000
EC01109=100.9998,0.0000
EC01110=102.5167,0.0000
EC01111=104.9212,0.0000
EC01112=107.8298,0.0000
EC01113=110.9268,0.0000
EC01114=114.0730,0.0000
EC01115=117.1707,0.0000
EC01116=120.0788,0.0000
EC01117=122.4830,0.0000
EC01118=124.0000,0.0000
EC01119=124.4140,0.0000
EC01120=124.6279,0.0000
EC01121=124.8952,0.0000
EC01122=125.4421,0.0000
EC01123=126.7764,0.0000
EC01124=129.5628,0.0000
EC01125=132.3404,0.0000
EC01126=135.0000,0.0000
EC01127=137.6596,0.0000
EC01128=140.4372,0.0000
EC01129=143.2236,0.0000
EC01130=144.5579,0.0000
EC01131=145.1048,0.0000
EC01132=145.3721,0.0000
EC01133=145.5860,0.0000
EC01134=146.0000,0.0000
EC01135=147.5170,0.0000
EC01136=149.9212,0.0000
EC01137=152.8293,0.0000
EC01138=155.9270,0.0000
EC01139=159.0732,0.0000
EC01140=162.1702,0.0000
EC01141=165.0788,0.0000
EC01142=167.4833,0.0000
EC01143=169.0002,0.0000
EC01144=169.4136,0.0000
EC01145=169.6281,0.0000
EC01146=169.8955,0.0000
EC01147=170.4423,0.0000
EC01148=171.7765,0.0000
EC01149=174.5632,0.0000
EC01150=177.3397,0.0000
EC01151=180.0000,0.0000
EC01152=180.0000,0.0000
EC01153=-177.3397,0.0000
EC01154=-174.5632,0.0000
EC01155=-171.7765,0.0000
EC01156=-170.4423,0.0000
EC01157=-169.8955,0.0000
EC01158=-169.6281,0.0000
EC01159=-169.4136,0.0000
EC01160=-169.0002,0.0000
EC01161=-167.4833,0.0000
EC01162=-165.0788,0.0000
EC01163=-162.1702,0.0000
EC01164=-159.0732,0.0000
EC01165=-155.9270,0.0000
EC01166=-152.8293,0.0000
EC01167=-149.9212,0.0000
EC01168=-147.5170,0.0000
EC01169=-146.0000,0.0000
EC01170=-145.5860,0.0000
EC01171=-145.3721,0.0000
EC01172=-145.1048,0.0000
EC01173=-144.5579,0.0000
EC01174=-143.2236,0.0000
EC01175=-140.4372,0.0000
EC01176=-137.6596,0.0000
EC01177=-135.0000,0.0000
EC01178=-132.3404,0.0000
EC01179=-129.5628,0.0000
EC01180=-126.7764,0.0000
EC01181=-125.4421,0.0000
EC01182=-124.8952,0.0000
EC01183=-124.6279,0.0000
EC01184=-124.4140,0.0000
EC01185=-124.0000,0.0000
EC01186=-122.4830,0.0000
EC01187=-120.0788,0.0000
EC01188=-117.1707,0.0000
EC01189=-114.0730,0.0000
EC01190=-110.9268,0.0000
EC01191=-107.8298,0.0000
EC01192=-104.9212,0.0000
EC01193=-102.5167,0.0000
EC01194=-100.9998,0.0000
EC01195=-100.5864,0.0000
EC01196=-100.3719,0.0000
EC01197=-100.1045,0.0000
EC01198=-99.5577,0.0000
EC01199=-98.2235,0.0000
EC01200=-95.4368,0.0000
EC01201=-92.6603,0.0000
EC01202=-90.0000,0.0000
EC01203=-87.3397,0.0000
EC01204=-84.5632,0.0000
EC01205=-81.7765,0.0000
EC01206=-80.4423,0.0000
EC01207=-79.8955,0.0000
EC01208=-79.6281,0.0000
EC01209=-79.4136,0.0000
EC01210=-79.0002,0.0000
EC01211=-77.4833,0.0000
EC01212=-75.0788,0.0000
EC01213=-72.1702,0.0000
EC01214=-69.0732,0.0000
EC01215=-65.9270,0.0000
EC01216=-62.8293,0.0000
EC01217=-59.9212,0.0000
EC01218=-57.5170,0.0000
EC01219=-56.0000,0.0000
EC01220=-55.5860,0.0000
EC01221=-55.3721,0.0000
EC01222=-55.1048,0.0000
EC01223=-54.5579,0.0000
EC01224=-53.2236,0.0000
EC01225=-50.4372,0.0000
EC01226=-47.6596,0.0000
EC01227=-45.0000,0.0000
EC01228=-42.3404,0.0000
EC01229=-39.5628,0.0000
EC01230=-36.7764,0.0000
EC01231=-35.4421,0.0000
EC01232=-34.8952,0.0000
EC01233=-34.6279,0.0000
EC01234=-34.4140,0.0000
EC01235=-34.0000,0.0000
EC01236=-32.4830,0.0000
EC01237=-30.0788,0.0000
EC01238=-27.1707,0.0000
EC01239=-24.0730,0.0000
EC01240=-20.9268,0.0000
EC01241=-17.8298,0.0000
EC01242=-14.9212,0.0000
EC01243=-12.5167,0.0000
EC01244=-10.9998,0.0000
EC01245=-10.5864,0.0000
EC01246=-10.3719,0.0000
EC01247=-10.1045,0.0000
EC01248=-9.5577,0.0000
EC01249=-8.2235,0.0000
EC01250=-5.4368,0.0000
EC01251=-2.6603,0.0000
EC01252=0.0000,0.0000
EC01253=0.0000,0.0000
EC01254=2.6105,0.0000
EC01255=5.3720,0.0000
EC01256=8.1701,0.0000
EC01257=9.4699,0.0000
EC01258=9.9705,0.0000
EC01259=10.1944,0.0000
EC01260=10.3679,0.0000
EC01261=10.7398,0.0000
EC01262=12.2618,0.0000
EC01263=14.7112,0.0000
EC01264=17.6927,0.0000
EC01265=20.8797,0.0000
EC01266=24.1202,0.0000
EC01267=27.3076,0.0000
EC01268=30.2891,0.0000
EC01269=32.7379,0.0000
EC01270=34.2600,0.0000
EC01271=34.6321,0.0000
EC01272=34.8056,0.0000
EC01273=35.0300,0.0000
EC01274=35.5299,0.0000
EC01275=36.8301,0.0000
EC01276=39.6279,0.0000
EC01277=42.3891,0.0000
EC01278=45.0000,0.0000
EC01279=47.6109,0.0000
EC01280=50.3721,0.0000
EC01281=53.1699,0.0000
EC01282=54.4701,0.0000
EC01283=54.9700,0.0000
EC01284=55.1944,0.0000
EC01285=55.3679,0.0000
EC01286=55.7400,0.0000
EC01287=57.2621,0.0000
EC01288=59.7109,0.0000
EC01289=62.6924,0.0000
EC01290=65.8798,0.0000
EC01291=69.1203,0.0000
EC01292=72.3073,0.0000
EC01293=75.2888,0.0000
EC01294=77.7382,0.0000
EC01295=79.2602,0.0000
EC01296=79.6321,0.0000
EC01297=79.8056,0.0000
EC01298=80.0295,0.0000
EC01299=80.5301,0.0000
EC01300=81.8299,0.0000
EC01301=84.6280,0.0000
EC01302=87.3895,0.0000
EC01303=90.0000,0.0000
EC01304=92.6105,0.0000
EC01305=95.3720,0.0000
EC01306=98.1701,0.0000
EC01307=99.4699,0.0000
EC01308=99.9705,0.0000
EC01309=100.1944,0.0000
EC01310=100.3679,0.0000
EC01311=100.7398,0.0000
EC01312=102.2618,0.0000
EC01313=104.7112,0.0000
EC01314=107.6927,0.0000
EC01315=110.8797,0.0000
EC01316=114.1202,0.0000
EC01317=117.3076,0.0000
EC01318=120.2891,0.0000
EC01319=122.7379,0.0000
EC01320=124.2600,0.0000
EC01321=124.6321,0.0000
EC01322=124.8056,0.0000
EC01323=125.0300,0.0000
EC01324=125.5299,0.0000
EC01325=126.8301,0.0000
EC01326=129.6279,0.0000
EC01327=132.3891,0.0000
EC01328=135.0000,0.0000
EC01329=137.6109,0.0000
EC01330=140.3721,0.0000
EC01331=143.1699,0.0000
EC01332=144.4701,0.0000
EC01333=144.9700,0.0000
EC01334=145.1944,0.0000
EC01335=145.3679,0.0000
EC01336=145.7400,0.0000
EC01337=147.2621,0.0000
EC01338=149.7109,0.0000
EC01339=152.6924,0.0000
EC01340=155.8798,0.0000
EC01341=159.1203,0.0000
EC01342=162.3073,0.0000
EC01343=165.2888,0.0000
EC01344=167.7382,0.0000
EC01345=169.2602,0.0000
EC01346=169.6321,0.0000
EC01347=169.8056,0.0000
EC01348=170.0295,0.0000
EC01349=170.5301,0.0000
EC01350=171.8299,0.0000
EC01351=174.6280,0.0000
EC01352=177.3895,0.0000
EC01353=180.0000,0.0000
EC01354=180.0000,0.0000
EC01355=-177.3895,0.0000
EC01356=-174.6280,0.0000
EC01357=-171.8299,0.0000
EC01358=-170.5301,0.0000
EC01359=-170.0295,0.0000
EC01360=-169.8056,0.0000
EC01361=-169.6321,0.0000
EC01362=-169.2602,0.0000
EC01363=-167.7382,0.0000
EC01364=-165.2888,0.0000
EC01365=-162.3073,0.0000
EC01366=-159.1203,0.0000
EC01367=-155.8798,0.0000
EC01368=-152.6924,0.0000
EC01369=-149.7109,0.0000
EC01370=-147.2621,0.0000
EC01371=-145.7400,0.0000
EC01372=-145.3679,0.0000
EC01373=-145.1944,0.0000
EC01374=-144.9700,0.0000
EC01375=-144.4701,0.0000
EC01376=-143.1699,0.0000
EC01377=-140.3721,0.0000
EC01378=-137.6109,0.0000
EC01379=-135.0000,0.0000
EC01380=-132.3891,0.0000
EC01381=-129.6279,0.0000
EC01382=-126.8301,0.0000
EC01383=-125.5299,0.0000
EC01384=-125.0300,0.0000
EC01385=-124.8056,0.0000
EC01386=-124.6321,0.0000
EC01387=-124.2600,0.0000
EC01388=-122.7379,0.0000
EC01389=-120.2891,0.0000
EC01390=-117.3076,0.0000
EC01391=-114.1202,0.0000
EC01392=-110.8797,0.0000
EC01393=-107.6927,0.0000
EC01394=-104.7112,0.0000
EC01395=-102.2618,0.0000
EC01396=-100.7398,0.0000
EC01397=-100.3679,0.0000
EC01398=-100.1944,0.0000
EC01399=-99.9705,0.0000
EC01400=-99.4699,0.0000
EC01401=-98.1701,0.0000
EC01402=-95.3720,0.0000
EC01403=-92.6105,0.0000
EC01404=-90.0000,0.0000
EC01405=-87.3895,0.0000
EC01406=-84.6280,0.0000
EC01407=-81.8299,0.0000
EC01408=-80.5301,0.0000
EC01409=-80.0295,0.0000
EC01410=-79.8056,0.0000
EC01411=-79.6321,0.0000
EC01412=-79.2602,0.0000
EC01413=-77.7382,0.0000
EC01414=-75.2888,0.0000
EC01415=-72.3073,0.0000
EC01416=-69.1203,0.0000
EC01417=-65.8798,0.0000
EC01418=-62.6924,0.0000
EC01419=-59.7109,0.0000
EC01420=-57.2621,0.0000
EC01421=-55.7400,0.0000
EC01422=-55.3679,0.0000
EC01423=-55.1944,0.0000
EC01424=-54.9700,0.0000
EC01425=-54.4701,0.0000
EC01426=-53.1699,0.0000
EC01427=-50.3721,0.0000
EC01428=-47.6109,0.0000
EC01429=-45.0000,0.0000
EC01430=-42.3891,0.0000
EC01431=-39.6279,0.0000
EC01432=-36.8301,0.0000
EC01433=-35.5299,0.0000
EC01434=-35.0300,0.0000
EC01435=-34.8056,0.0000
EC01436=-34.6321,0.0000
EC01437=-34.2600,0.0000
EC01438=-32.7379,0.0000
EC01439=-30.2891,0.0000
EC01440=-27.3076,0.0000
EC01441=-24.1202,0.0000
EC01442=-20.8797,0.0000
EC01443=-17.6927,0.0000
EC01444=-14.7112,0.0000
EC01445=-12.2618,0.0000
EC01446=-10.7398,0.0000
EC01447=-10.3679,0.0000
EC01448=-10.1944,0.0000
EC01449=-9.9705,0.0000
EC01450=-9.4699,0.0000
EC01451=-8.1701,0.0000
EC01452=-5.3720,0.0000
EC01453=-2.6105,0.0000
EC01454=0.0000,0.0000
EC01455=0.0000,0.0000
EC01456=2.5595,0.0000
EC01457=5.3045,0.0000
EC01458=8.1135,0.0000
EC01459=9.3788,0.0000
EC01460=9.8327,0.0000
EC01461=10.0151,0.0000
EC01462=10.1489,0.0000
EC01463=10.4816,0.0000
EC01464=12.0102,0.0000
EC01465=14.5040,0.0000
EC01466=17.5575,0.0000
EC01467=20.8329,0.0000
EC01468=24.1669,0.0000
EC01469=27.4422,0.0000
EC01470=30.4960,0.0000
EC01471=32.9901,0.0000
EC01472=34.5184,0.0000
EC01473=34.8513,0.0000
EC01474=34.9851,0.0000
EC01475=35.1672,0.0000
EC01476=35.6212,0.0000
EC01477=36.8860,0.0000
EC01478=39.6950,0.0000
EC01479=42.4397,0.0000
EC01480=45.0000,0.0000
EC01481=47.5591,0.0000
EC01482=50.3050,0.0000
EC01483=53.1140,0.0000
EC01484=54.3788,0.0000
EC01485=54.8328,0.0000
EC01486=55.0149,0.0000
EC01487=55.1487,0.0000
EC01488=55.4816,0.0000
EC01489=57.0099,0.0000
EC01490=59.5040,0.0000
EC01491=62.5578,0.0000
EC01492=65.8331,0.0000
EC01493=69.1671,0.0000
EC01494=72.4425,0.0000
EC01495=75.4960,0.0000
EC01496=77.9898,0.0000
EC01497=79.5184,0.0000
EC01498=79.8511,0.0000
EC01499=79.9849,0.0000
EC01500=80.1673,0.0000
EC01501=80.6212,0.0000
EC01502=81.8865,0.0000
EC01503=84.6955,0.0000
EC01504=87.4405,0.0000
EC01505=90.0000,0.0000
EC01506=92.5595,0.0000
EC01507=95.3053,0.0000
EC01508=98.1143,0.0000
EC01509=99.3788,0.0000
EC01510=99.8327,0.0000
EC01511=100.0151,0.0000
EC01512=100.1489,0.0000
EC01513=100.4816,0.0000
EC01514=102.0102,0.0000
EC01515=104.5040,0.0000
EC01516=107.5575,0.0000
EC01517=110.8329,0.0000
EC01518=114.1669,0.0000
EC01519=117.4422,0.0000
EC01520=120.4960,0.0000
EC01521=122.9901,0.0000
EC01522=124.5184,0.0000
EC01523=124.8513,0.0000
EC01524=124.9851,0.0000
EC01525=125.1672,0.0000
EC01526=125.6212,0.0000
EC01527=126.8860,0.0000
EC01528=129.6950,0.0000
EC01529=132.4397,0.0000
EC01530=135.0000,0.0000
EC01531=137.5591,0.0000
EC01532=140.3050,0.0000
EC01533=143.1140,0.0000
EC01534=144.3788,0.0000
EC01535=144.8328,0.0000
EC01536=145.0149,0.0000
EC01537=145.1487,0.0000
EC01538=145.4816,0.0000
EC01539=147.0099,0.0000
EC01540=149.5040,0.0000
EC01541=152.5578,0.0000
EC01542=155.8331,0.0000
EC01543=159.1671,0.0000
EC01544=162.4425,0.0000
EC01545=165.4960,0.0000
EC01546=167.9898,0.0000
EC01547=169.5184,0.0000
EC01548=169.8511,0.0000
EC01549=169.9849,0.0000
EC01550=170.1673,0.0000
EC01551=170.6212,0.0000
EC01552=171.8865,0.0000
EC01553=174.6955,0.0000
EC01554=177.4405,0.0000
EC01555=180.0000,0.0000
EC01556=180.0000,0.0000
EC01557=-177.4405,0.0000
EC01558=-174.6947,0.0000
EC01559=-171.8857,0.0000
EC01560=-170.6212,0.0000
EC01561=-170.1673,0.0000
EC01562=-169.9849,0.0000
EC01563=-169.8511,0.0000
EC01564=-169.5184,0.0000
EC01565=-167.9898,0.0000
EC01566=-165.4960,0.0000
EC01567=-162.4425,0.0000
EC01568=-159.1671,0.0000
EC01569=-155.8331,0.0000
EC01570=-152.5578,0.0000
EC01571=-149.5040,0.0000
EC01572=-147.0099,0.0000
EC01573=-145.4816,0.0000
EC01574=-145.1487,0.0000
EC01575=-145.0149,0.0000
EC01576=-144.8328,0.0000
EC01577=-144.3788,0.0000
EC01578=-143.1140,0.0000
EC01579=-140.3050,0.0000
EC01580=-137.5603,0.0000
EC01581=-135.0000,0.0000
EC01582=-132.4409,0.0000
EC01583=-129.6950,0.0000
EC01584=-126.8860,0.0000
EC01585=-125.6212,0.0000
EC01586=-125.1672,0.0000
EC01587=-124.9851,0.0000
EC01588=-124.8513,0.0000
EC01589=-124.5184,0.0000
EC01590=-122.9901,0.0000
EC01591=-120.4960,0.0000
EC01592=-117.4422,0.0000
EC01593=-114.1669,0.0000
EC01594=-110.8329,0.0000
EC01595=-107.5575,0.0000
EC01596=-104.5040,0.0000
EC01597=-102.0102,0.0000
EC01598=-100.4816,0.0000
EC01599=-100.1489,0.0000
EC01600=-100.0151,0.0000
EC01601=-99.8327,0.0000
EC01602=-99.3788,0.0000
EC01603=-98.1135,0.0000
EC01604=-95.3045,0.0000
EC01605=-92.5595,0.0000
EC01606=-90.0000,0.0000
EC01607=-87.4405,0.0000
EC01608=-84.6947,0.0000
EC01609=-81.8857,0.0000
EC01610=-80.6212,0.0000
EC01611=-80.1673,0.0000
EC01612=-79.9849,0.0000
EC01613=-79.8511,0.0000
EC01614=-79.5184,0.0000
EC01615=-77.9898,0.0000
EC01616=-75.4960,0.0000
EC01617=-72.4425,0.0000
EC01618=-69.1671,0.0000
EC01619=-65.8331,0.0000
EC01620=-62.5578,0.0000
EC01621=-59.5040,0.0000
EC01622=-57.0099,0.0000
EC01623=-55.4816,0.0000
EC01624=-55.1487,0.0000
EC01625=-55.0149,0.0000
EC01626=-54.8328,0.0000
EC01627=-54.3788,0.0000
EC01628=-53.1140,0.0000
EC01629=-50.3050,0.0000
EC01630=-47.5603,0.0000
EC01631=-45.0000,0.0000
EC01632=-42.4409,0.0000
EC01633=-39.6950,0.0000
EC01634=-36.8860,0.0000
EC01635=-35.6212,0.0000
EC01636=-35.1672,0.0000
EC01637=-34.9851,0.0000
EC01638=-34.8513,0.0000
EC01639=-34.5184,0.0000
EC01640=-32.9901,0.0000
EC01641=-30.4960,0.0000
EC01642=-27.4422,0.0000
EC01643=-24.1669,0.0000
EC01644=-20.8329,0.0000
EC01645=-17.5575,0.0000
EC01646=-14.5040,0.0000
EC01647=-12.0102,0.0000
EC01648=-10.4816,0.0000
EC01649=-10.1489,0.0000
EC01650=-10.0151,0.0000
EC01651=-9.8327,0.0000
EC01652=-9.3788,0.0000
EC01653=-8.1143,0.0000
EC01654=-5.3053,0.0000
EC01655=-2.5595,0.0000
EC01656=0.0000,0.0000
EC01657=0.0000,0.0000
EC01658=2.5072,0.0000
EC01659=5.2349,0.0000
EC01660=8.0561,0.0000
EC01661=9.2852,0.0000
EC01662=9.6930,0.0000
EC01663=9.8344,0.0000
EC01664=9.9312,0.0000
EC01665=10.2265,0.0000
EC01666=11.7624,0.0000
EC01667=14.3014,0.0000
EC01668=17.4259,0.0000
EC01669=20.7876,0.0000
EC01670=24.2123,0.0000
EC01671=27.5744,0.0000
EC01672=30.6985,0.0000
EC01673=33.2374,0.0000
EC01674=34.7737,0.0000
EC01675=35.0694,0.0000
EC01676=35.1660,0.0000
EC01677=35.3073,0.0000
EC01678=35.7148,0.0000
EC01679=36.9441,0.0000
EC01680=39.7651,0.0000
EC01681=42.4931,0.0000
EC01682=45.0000,0.0000
EC01683=47.5069,0.0000
EC01684=50.2349,0.0000
EC01685=53.0566,0.0000
EC01686=54.2852,0.0000
EC01687=54.6927,0.0000
EC01688=54.8340,0.0000
EC01689=54.9306,0.0000
EC01690=55.2263,0.0000
EC01691=56.7626,0.0000
EC01692=59.3015,0.0000
EC01693=62.4256,0.0000
EC01694=65.7877,0.0000
EC01695=69.2124,0.0000
EC01696=72.5741,0.0000
EC01697=75.6986,0.0000
EC01698=78.2376,0.0000
EC01699=79.7735,0.0000
EC01700=80.0688,0.0000
EC01701=80.1656,0.0000
EC01702=80.3070,0.0000
EC01703=80.7148,0.0000
EC01704=81.9439,0.0000
EC01705=84.7651,0.0000
EC01706=87.4928,0.0000
EC01707=90.0000,0.0000
EC01708=92.5064,0.0000
EC01709=95.2349,0.0000
EC01710=98.0561,0.0000
EC01711=99.2852,0.0000
EC01712=99.6930,0.0000
EC01713=99.8344,0.0000
EC01714=99.9312,0.0000
EC01715=100.2265,0.0000
EC01716=101.7624,0.0000
EC01717=104.3014,0.0000
EC01718=107.4259,0.0000
EC01719=110.7876,0.0000
EC01720=114.2123,0.0000
EC01721=117.5744,0.0000
EC01722=120.6985,0.0000
EC01723=123.2374,0.0000
EC01724=124.7737,0.0000
EC01725=125.0694,0.0000
EC01726=125.1660,0.0000
EC01727=125.3073,0.0000
EC01728=125.7148,0.0000
EC01729=126.9441,0.0000
EC01730=129.7651,0.0000
EC01731=132.4931,0.0000
EC01732=135.0000,0.0000
EC01733=137.5069,0.0000
EC01734=140.2349,0.0000
EC01735=143.0566,0.0000
EC01736=144.2852,0.0000
EC01737=144.6927,0.0000
EC01738=144.8340,0.0000
EC01739=144.9306,0.0000
EC01740=145.2263,0.0000
EC01741=146.7626,0.0000
EC01742=149.3015,0.0000
EC01743=152.4256,0.0000
EC01744=155.7877,0.0000
EC01745=159.2124,0.0000
EC01746=162.5741,0.0000
EC01747=165.6986,0.0000
EC01748=168.2376,0.0000
EC01749=169.7735,0.0000
EC01750=170.0688,0.0000
EC01751=170.1656,0.0000
EC01752=170.3070,0.0000
EC01753=170.7148,0.0000
EC01754=171.9439,0.0000
EC01755=174.7651,0.0000
EC01756=177.4928,0.0000
EC01757=180.0000,0.0000
EC01758=180.0000,0.0000
EC01759=-177.4936,0.0000
EC01760=-174.7651,0.0000
EC01761=-171.9439,0.0000
EC01762=-170.7148,0.0000
EC01763=-170.3070,0.0000
EC01764=-170.1656,0.0000
EC01765=-170.0688,0.0000
EC01766=-169.7735,0.0000
EC01767=-168.2376,0.0000
EC01768=-165.6986,0.0000
EC01769=-162.5741,0.0000
EC01770=-159.2124,0.0000
EC01771=-155.7877,0.0000
EC01772=-152.4256,0.0000
EC01773=-149.3015,0.0000
EC01774=-146.7626,0.0000
EC01775=-145.2263,0.0000
EC01776=-144.9306,0.0000
EC01777=-144.8340,0.0000
EC01778=-144.6927,0.0000
EC01779=-144.2852,0.0000
EC01780=-143.0559,0.0000
EC01781=-140.2349,0.0000
EC01782=-137.5069,0.0000
EC01783=-135.0000,0.0000
EC01784=-132.4931,0.0000
EC01785=-129.7651,0.0000
EC01786=-126.9434,0.0000
EC01787=-125.7148,0.0000
EC01788=-125.3073,0.0000
EC01789=-125.1660,0.0000
EC01790=-125.0694,0.0000
EC01791=-124.7737,0.0000
EC01792=-123.2374,0.0000
EC01793=-120.6985,0.0000
EC01794=-117.5744,0.0000
EC01795=-114.2123,0.0000
EC01796=-110.7876,0.0000
EC01797=-107.4259,0.0000
EC01798=-104.3014,0.0000
EC01799=-101.7624,0.0000
EC01800=-100.2265,0.0000
EC01801=-99.9312,0.0000
EC01802=-99.8344,0.0000
EC01803=-99.6930,0.0000
EC01804=-99.2852,0.0000
EC01805=-98.0561,0.0000
EC01806=-95.2349,0.0000
EC01807=-92.5072,0.0000
EC01808=-90.0000,0.0000
EC01809=-87.4936,0.0000
EC01810=-84.7651,0.0000
EC01811=-81.9439,0.0000
EC01812=-80.7148,0.0000
EC01813=-80.3070,0.0000
EC01814=-80.1656,0.0000
EC01815=-80.0688,0.0000
EC01816=-79.7735,0.0000
EC01817=-78.2376,0.0000
EC01818=-75.6986,0.0000
EC01819=-72.5741,0.0000
EC01820=-69.2124,0.0000
EC01821=-65.7877,0.0000
EC01822=-62.4256,0.0000
EC01823=-59.3015,0.0000
EC01824=-56.7626,0.0000
EC01825=-55.2263,0.0000
EC01826=-54.9306,0.0000
EC01827=-54.8340,0.0000
EC01828=-54.6927,0.0000
EC01829=-54.2852,0.0000
EC01830=-53.0559,0.0000
EC01831=-50.2349,0.0000
EC01832=-47.5069,0.0000
EC01833=-45.0000,0.0000
EC01834=-42.4931,0.0000
EC01835=-39.7651,0.0000
EC01836=-36.9434,0.0000
EC01837=-35.7148,0.0000
EC01838=-35.3073,0.0000
EC01839=-35.1660,0.0000
EC01840=-35.0694,0.0000
EC01841=-34.7737,0.0000
EC01842=-33.2374,0.0000
EC01843=-30.6985,0.0000
EC01844=-27.5744,0.0000
EC01845=-24.2123,0.0000
EC01846=-20.7876,0.0000
EC01847=-17.4259,0.0000
EC01848=-14.3014,0.0000
EC01849=-11.7624,0.0000
EC01850=-10.2265,0.0000
EC01851=-9.9312,0.0000
EC01852=-9.8344,0.0000
EC01853=-9.6930,0.0000
EC01854=-9.2852,0.0000
EC01855=-8.0561,0.0000
EC01856=-5.2349,0.0000
EC01857=-2.5064,0.0000
EC01858=0.0000,0.0000
EC01859=0.0000,0.0000
EC01860=2.4517,0.0000
EC01861=5.1629,0.0000
EC01862=7.9963,0.0000
EC01863=9.1897,0.0000
EC01864=9.5501,0.0000
EC01865=9.6525,0.0000
EC01866=9.7146,0.0000
EC01867=9.9757,0.0000
EC01868=11.5206,0.0000
EC01869=14.1038,0.0000
EC01870=17.2974,0.0000
EC01871=20.7433,0.0000
EC01872=24.2566,0.0000
EC01873=27.7026,0.0000
EC01874=30.8962,0.0000
EC01875=33.4793,0.0000
EC01876=35.0245,0.0000
EC01877=35.2855,0.0000
EC01878=35.3476,0.0000
EC01879=35.4495,0.0000
EC01880=35.8105,0.0000
EC01881=37.0038,0.0000
EC01882=39.8372,0.0000
EC01883=42.5482,0.0000
EC01884=45.0000,0.0000
EC01885=47.4518,0.0000
EC01886=50.1628,0.0000
EC01887=52.9966,0.0000
EC01888=54.1895,0.0000
EC01889=54.5505,0.0000
EC01890=54.6524,0.0000
EC01891=54.7145,0.0000
EC01892=54.9755,0.0000
EC01893=56.5207,0.0000
EC01894=59.1038,0.0000
EC01895=62.2974,0.0000
EC01896=65.7434,0.0000
EC01897=69.2567,0.0000
EC01898=72.7026,0.0000
EC01899=75.8962,0.0000
EC01900=78.4794,0.0000
EC01901=80.0243,0.0000
EC01902=80.2854,0.0000
EC01903=80.3475,0.0000
EC01904=80.4499,0.0000
EC01905=80.8103,0.0000
EC01906=82.0037,0.0000
EC01907=84.8371,0.0000
EC01908=87.5483,0.0000
EC01909=90.0000,0.0000
EC01910=92.4517,0.0000
EC01911=95.1629,0.0000
EC01912=97.9963,0.0000
EC01913=99.1897,0.0000
EC01914=99.5501,0.0000
EC01915=99.6525,0.0000
EC01916=99.7146,0.0000
EC01917=99.9757,0.0000
EC01918=101.5206,0.0000
EC01919=104.1038,0.0000
EC01920=107.2974,0.0000
EC01921=110.7433,0.0000
EC01922=114.2566,0.0000
EC01923=117.7026,0.0000
EC01924=120.8962,0.0000
EC01925=123.4793,0.0000
EC01926=125.0245,0.0000
EC01927=125.2855,0.0000
EC01928=125.3476,0.0000
EC01929=125.4495,0.0000
EC01930=125.8105,0.0000
EC01931=127.0038,0.0000
EC01932=129.8372,0.0000
EC01933=132.5482,0.0000
EC01934=135.0000,0.0000
EC01935=137.4518,0.0000
EC01936=140.1628,0.0000
EC01937=142.9966,0.0000
EC01938=144.1895,0.0000
EC01939=144.5505,0.0000
EC01940=144.6524,0.0000
EC01941=144.7145,0.0000
EC01942=144.9755,0.0000
EC01943=146.5207,0.0000
EC01944=149.1038,0.0000
EC01945=152.2974,0.0000
EC01946=155.7434,0.0000
EC01947=159.2567,0.0000
EC01948=162.7026,0.0000
EC01949=165.8962,0.0000
EC01950=168.4794,0.0000
EC01951=170.0243,0.0000
EC01952=170.2854,0.0000
EC01953=170.3475,0.0000
EC01954=170.4499,0.0000
EC01955=170.8103,0.0000
EC01956=172.0037,0.0000
EC01957=174.8371,0.0000
EC01958=177.5483,0.0000
EC01959=180.0000,0.0000
EC01960=180.0000,0.0000
EC01961=-177.5483,0.0000
EC01962=-174.8371,0.0000
EC01963=-172.0037,0.0000
EC01964=-170.8103,0.0000
EC01965=-170.4499,0.0000
EC01966=-170.3475,0.0000
EC01967=-170.2854,0.0000
EC01968=-170.0243,0.0000
EC01969=-168.4794,0.0000
EC01970=-165.8962,0.0000
EC01971=-162.7026,0.0000
EC01972=-159.2567,0.0000
EC01973=-155.7434,0.0000
EC01974=-152.2974,0.0000
EC01975=-149.1038,0.0000
EC01976=-146.5207,0.0000
EC01977=-144.9755,0.0000
EC01978=-144.7145,0.0000
EC01979=-144.6524,0.0000
EC01980=-144.5505,0.0000
EC01981=-144.1895,0.0000
EC01982=-142.9962,0.0000
EC01983=-140.1628,0.0000
EC01984=-137.4518,0.0000
EC01985=-135.0000,0.0000
EC01986=-132.5482,0.0000
EC01987=-129.8372,0.0000
EC01988=-127.0034,0.0000
EC01989=-125.8105,0.0000
EC01990=-125.4495,0.0000
EC01991=-125.3476,0.0000
EC01992=-125.2855,0.0000
EC01993=-125.0245,0.0000
EC01994=-123.4793,0.0000
EC01995=-120.8962,0.0000
EC01996=-117.7026,0.0000
EC01997=-114.2566,0.0000
EC01998=-110.7433,0.0000
EC01999=-107.2974,0.0000
//INST
///DATE 2021/02/10 13:51
///COMM
///ATTR SC,RW,RJ
////FRAME USER 2
///GROUP1 RB1
///GROUP2 ST1
NOP
SMOVL C00000 +MOVJ EC00000
SMOVL C00001 +MOVJ EC00001
SMOVL C00002 +MOVJ EC00002
SMOVL C00003 +MOVJ EC00003
SMOVL C00004 +MOVJ EC00004
SMOVL C00005 +MOVJ EC00005
SMOVL C00006 +MOVJ EC00006
SMOVL C00007 +MOVJ EC00007
SMOVL C00008 +MOVJ EC00008
SMOVL C00009 +MOVJ EC00009
SMOVL C00010 +MOVJ EC00010
SMOVL C00011 +MOVJ EC00011
SMOVL C00012 +MOVJ EC00012
SMOVL C00013 +MOVJ EC00013
SMOVL C00014 +MOVJ EC00014
SMOVL C00015 +MOVJ EC00015
SMOVL C00016 +MOVJ EC00016
SMOVL C00017 +MOVJ EC00017
SMOVL C00018 +MOVJ EC00018
SMOVL C00019 +MOVJ EC00019
SMOVL C00020 +MOVJ EC00020
SMOVL C00021 +MOVJ EC00021
SMOVL C00022 +MOVJ EC00022
SMOVL C00023 +MOVJ EC00023
SMOVL C00024 +MOVJ EC00024
SMOVL C00025 +MOVJ EC00025
SMOVL C00026 +MOVJ EC00026
SMOVL C00027 +MOVJ EC00027
SMOVL C00028 +MOVJ EC00028
SMOVL C00029 +MOVJ EC00029
SMOVL C00030 +MOVJ EC00030
SMOVL C00031 +MOVJ EC00031
SMOVL C00032 +MOVJ EC00032
SMOVL C00033 +MOVJ EC00033
SMOVL C00034 +MOVJ EC00034
SMOVL C00035 +MOVJ EC00035
SMOVL C00036 +MOVJ EC00036
SMOVL C00037 +MOVJ EC00037
SMOVL C00038 +MOVJ EC00038
SMOVL C00039 +MOVJ EC00039
SMOVL C00040 +MOVJ EC00040
SMOVL C00041 +MOVJ EC00041
SMOVL C00042 +MOVJ EC00042
SMOVL C00043 +MOVJ EC00043
SMOVL C00044 +MOVJ EC00044
SMOVL C00045 +MOVJ EC00045
SMOVL C00046 +MOVJ EC00046
SMOVL C00047 +MOVJ EC00047
SMOVL C00048 +MOVJ EC00048
SMOVL C00049 +MOVJ EC00049
SMOVL C00050 +MOVJ EC00050
SMOVL C00051 +MOVJ EC00051
SMOVL C00052 +MOVJ EC00052
SMOVL C00053 +MOVJ EC00053
SMOVL C00054 +MOVJ EC00054
SMOVL C00055 +MOVJ EC00055
SMOVL C00056 +MOVJ EC00056
SMOVL C00057 +MOVJ EC00057
SMOVL C00058 +MOVJ EC00058
SMOVL C00059 +MOVJ EC00059
SMOVL C00060 +MOVJ EC00060
SMOVL C00061 +MOVJ EC00061
SMOVL C00062 +MOVJ EC00062
SMOVL C00063 +MOVJ EC00063
SMOVL C00064 +MOVJ EC00064
SMOVL C00065 +MOVJ EC00065
SMOVL C00066 +MOVJ EC00066
SMOVL C00067 +MOVJ EC00067
SMOVL C00068 +MOVJ EC00068
SMOVL C00069 +MOVJ EC00069
SMOVL C00070 +MOVJ EC00070
SMOVL C00071 +MOVJ EC00071
SMOVL C00072 +MOVJ EC00072
SMOVL C00073 +MOVJ EC00073
SMOVL C00074 +MOVJ EC00074
SMOVL C00075 +MOVJ EC00075
SMOVL C00076 +MOVJ EC00076
SMOVL C00077 +MOVJ EC00077
SMOVL C00078 +MOVJ EC00078
SMOVL C00079 +MOVJ EC00079
SMOVL C00080 +MOVJ EC00080
SMOVL C00081 +MOVJ EC00081
SMOVL C00082 +MOVJ EC00082
SMOVL C00083 +MOVJ EC00083
SMOVL C00084 +MOVJ EC00084
SMOVL C00085 +MOVJ EC00085
SMOVL C00086 +MOVJ EC00086
SMOVL C00087 +MOVJ EC00087
SMOVL C00088 +MOVJ EC00088
SMOVL C00089 +MOVJ EC00089
SMOVL C00090 +MOVJ EC00090
SMOVL C00091 +MOVJ EC00091
SMOVL C00092 +MOVJ EC00092
SMOVL C00093 +MOVJ EC00093
SMOVL C00094 +MOVJ EC00094
SMOVL C00095 +MOVJ EC00095
SMOVL C00096 +MOVJ EC00096
SMOVL C00097 +MOVJ EC00097
SMOVL C00098 +MOVJ EC00098
SMOVL C00099 +MOVJ EC00099
SMOVL C00100 +MOVJ EC00100
SMOVL C00101 +MOVJ EC00101
SMOVL C00102 +MOVJ EC00102
SMOVL C00103 +MOVJ EC00103
SMOVL C00104 +MOVJ EC00104
SMOVL C00105 +MOVJ EC00105
SMOVL C00106 +MOVJ EC00106
SMOVL C00107 +MOVJ EC00107
SMOVL C00108 +MOVJ EC00108
SMOVL C00109 +MOVJ EC00109
SMOVL C00110 +MOVJ EC00110
SMOVL C00111 +MOVJ EC00111
SMOVL C00112 +MOVJ EC00112
SMOVL C00113 +MOVJ EC00113
SMOVL C00114 +MOVJ EC00114
SMOVL C00115 +MOVJ EC00115
SMOVL C00116 +MOVJ EC00116
SMOVL C00117 +MOVJ EC00117
SMOVL C00118 +MOVJ EC00118
SMOVL C00119 +MOVJ EC00119
SMOVL C00120 +MOVJ EC00120
SMOVL C00121 +MOVJ EC00121
SMOVL C00122 +MOVJ EC00122
SMOVL C00123 +MOVJ EC00123
SMOVL C00124 +MOVJ EC00124
SMOVL C00125 +MOVJ EC00125
SMOVL C00126 +MOVJ EC00126
SMOVL C00127 +MOVJ EC00127
SMOVL C00128 +MOVJ EC00128
SMOVL C00129 +MOVJ EC00129
SMOVL C00130 +MOVJ EC00130
SMOVL C00131 +MOVJ EC00131
SMOVL C00132 +MOVJ EC00132
SMOVL C00133 +MOVJ EC00133
SMOVL C00134 +MOVJ EC00134
SMOVL C00135 +MOVJ EC00135
SMOVL C00136 +MOVJ EC00136
SMOVL C00137 +MOVJ EC00137
SMOVL C00138 +MOVJ EC00138
SMOVL C00139 +MOVJ EC00139
SMOVL C00140 +MOVJ EC00140
SMOVL C00141 +MOVJ EC00141
SMOVL C00142 +MOVJ EC00142
SMOVL C00143 +MOVJ EC00143
SMOVL C00144 +MOVJ EC00144
SMOVL C00145 +MOVJ EC00145
SMOVL C00146 +MOVJ EC00146
SMOVL C00147 +MOVJ EC00147
SMOVL C00148 +MOVJ EC00148
SMOVL C00149 +MOVJ EC00149
SMOVL C00150 +MOVJ EC00150
SMOVL C00151 +MOVJ EC00151
SMOVL C00152 +MOVJ EC00152
SMOVL C00153 +MOVJ EC00153
SMOVL C00154 +MOVJ EC00154
SMOVL C00155 +MOVJ EC00155
SMOVL C00156 +MOVJ EC00156
SMOVL C00157 +MOVJ EC00157
SMOVL C00158 +MOVJ EC00158
SMOVL C00159 +MOVJ EC00159
SMOVL C00160 +MOVJ EC00160
SMOVL C00161 +MOVJ EC00161
SMOVL C00162 +MOVJ EC00162
SMOVL C00163 +MOVJ EC00163
SMOVL C00164 +MOVJ EC00164
SMOVL C00165 +MOVJ EC00165
SMOVL C00166 +MOVJ EC00166
SMOVL C00167 +MOVJ EC00167
SMOVL C00168 +MOVJ EC00168
SMOVL C00169 +MOVJ EC00169
SMOVL C00170 +MOVJ EC00170
SMOVL C00171 +MOVJ EC00171
SMOVL C00172 +MOVJ EC00172
SMOVL C00173 +MOVJ EC00173
SMOVL C00174 +MOVJ EC00174
SMOVL C00175 +MOVJ EC00175
SMOVL C00176 +MOVJ EC00176
SMOVL C00177 +MOVJ EC00177
SMOVL C00178 +MOVJ EC00178
SMOVL C00179 +MOVJ EC00179
SMOVL C00180 +MOVJ EC00180
SMOVL C00181 +MOVJ EC00181
SMOVL C00182 +MOVJ EC00182
SMOVL C00183 +MOVJ EC00183
SMOVL C00184 +MOVJ EC00184
SMOVL C00185 +MOVJ EC00185
SMOVL C00186 +MOVJ EC00186
SMOVL C00187 +MOVJ EC00187
SMOVL C00188 +MOVJ EC00188
SMOVL C00189 +MOVJ EC00189
SMOVL C00190 +MOVJ EC00190
SMOVL C00191 +MOVJ EC00191
SMOVL C00192 +MOVJ EC00192
SMOVL C00193 +MOVJ EC00193
SMOVL C00194 +MOVJ EC00194
SMOVL C00195 +MOVJ EC00195
SMOVL C00196 +MOVJ EC00196
SMOVL C00197 +MOVJ EC00197
SMOVL C00198 +MOVJ EC00198
SMOVL C00199 +MOVJ EC00199
SMOVL C00200 +MOVJ EC00200
SMOVL C00201 +MOVJ EC00201
SMOVL C00202 +MOVJ EC00202
SMOVL C00203 +MOVJ EC00203
SMOVL C00204 +MOVJ EC00204
SMOVL C00205 +MOVJ EC00205
SMOVL C00206 +MOVJ EC00206
SMOVL C00207 +MOVJ EC00207
SMOVL C00208 +MOVJ EC00208
SMOVL C00209 +MOVJ EC00209
SMOVL C00210 +MOVJ EC00210
SMOVL C00211 +MOVJ EC00211
SMOVL C00212 +MOVJ EC00212
SMOVL C00213 +MOVJ EC00213
SMOVL C00214 +MOVJ EC00214
SMOVL C00215 +MOVJ EC00215
SMOVL C00216 +MOVJ EC00216
SMOVL C00217 +MOVJ EC00217
SMOVL C00218 +MOVJ EC00218
SMOVL C00219 +MOVJ EC00219
SMOVL C00220 +MOVJ EC00220
SMOVL C00221 +MOVJ EC00221
SMOVL C00222 +MOVJ EC00222
SMOVL C00223 +MOVJ EC00223
SMOVL C00224 +MOVJ EC00224
SMOVL C00225 +MOVJ EC00225
SMOVL C00226 +MOVJ EC00226
SMOVL C00227 +MOVJ EC00227
SMOVL C00228 +MOVJ EC00228
SMOVL C00229 +MOVJ EC00229
SMOVL C00230 +MOVJ EC00230
SMOVL C00231 +MOVJ EC00231
SMOVL C00232 +MOVJ EC00232
SMOVL C00233 +MOVJ EC00233
SMOVL C00234 +MOVJ EC00234
SMOVL C00235 +MOVJ EC00235
SMOVL C00236 +MOVJ EC00236
SMOVL C00237 +MOVJ EC00237
SMOVL C00238 +MOVJ EC00238
SMOVL C00239 +MOVJ EC00239
SMOVL C00240 +MOVJ EC00240
SMOVL C00241 +MOVJ EC00241
SMOVL C00242 +MOVJ EC00242
SMOVL C00243 +MOVJ EC00243
SMOVL C00244 +MOVJ EC00244
SMOVL C00245 +MOVJ EC00245
SMOVL C00246 +MOVJ EC00246
SMOVL C00247 +MOVJ EC00247
SMOVL C00248 +MOVJ EC00248
SMOVL C00249 +MOVJ EC00249
SMOVL C00250 +MOVJ EC00250
SMOVL C00251 +MOVJ EC00251
SMOVL C00252 +MOVJ EC00252
SMOVL C00253 +MOVJ EC00253
SMOVL C00254 +MOVJ EC00254
SMOVL C00255 +MOVJ EC00255
SMOVL C00256 +MOVJ EC00256
SMOVL C00257 +MOVJ EC00257
SMOVL C00258 +MOVJ EC00258
SMOVL C00259 +MOVJ EC00259
SMOVL C00260 +MOVJ EC00260
SMOVL C00261 +MOVJ EC00261
SMOVL C00262 +MOVJ EC00262
SMOVL C00263 +MOVJ EC00263
SMOVL C00264 +MOVJ EC00264
SMOVL C00265 +MOVJ EC00265
SMOVL C00266 +MOVJ EC00266
SMOVL C00267 +MOVJ EC00267
SMOVL C00268 +MOVJ EC00268
SMOVL C00269 +MOVJ EC00269
SMOVL C00270 +MOVJ EC00270
SMOVL C00271 +MOVJ EC00271
SMOVL C00272 +MOVJ EC00272
SMOVL C00273 +MOVJ EC00273
SMOVL C00274 +MOVJ EC00274
SMOVL C00275 +MOVJ EC00275
SMOVL C00276 +MOVJ EC00276
SMOVL C00277 +MOVJ EC00277
SMOVL C00278 +MOVJ EC00278
SMOVL C00279 +MOVJ EC00279
SMOVL C00280 +MOVJ EC00280
SMOVL C00281 +MOVJ EC00281
SMOVL C00282 +MOVJ EC00282
SMOVL C00283 +MOVJ EC00283
SMOVL C00284 +MOVJ EC00284
SMOVL C00285 +MOVJ EC00285
SMOVL C00286 +MOVJ EC00286
SMOVL C00287 +MOVJ EC00287
SMOVL C00288 +MOVJ EC00288
SMOVL C00289 +MOVJ EC00289
SMOVL C00290 +MOVJ EC00290
SMOVL C00291 +MOVJ EC00291
SMOVL C00292 +MOVJ EC00292
SMOVL C00293 +MOVJ EC00293
SMOVL C00294 +MOVJ EC00294
SMOVL C00295 +MOVJ EC00295
SMOVL C00296 +MOVJ EC00296
SMOVL C00297 +MOVJ EC00297
SMOVL C00298 +MOVJ EC00298
SMOVL C00299 +MOVJ EC00299
SMOVL C00300 +MOVJ EC00300
SMOVL C00301 +MOVJ EC00301
SMOVL C00302 +MOVJ EC00302
SMOVL C00303 +MOVJ EC00303
SMOVL C00304 +MOVJ EC00304
SMOVL C00305 +MOVJ EC00305
SMOVL C00306 +MOVJ EC00306
SMOVL C00307 +MOVJ EC00307
SMOVL C00308 +MOVJ EC00308
SMOVL C00309 +MOVJ EC00309
SMOVL C00310 +MOVJ EC00310
SMOVL C00311 +MOVJ EC00311
SMOVL C00312 +MOVJ EC00312
SMOVL C00313 +MOVJ EC00313
SMOVL C00314 +MOVJ EC00314
SMOVL C00315 +MOVJ EC00315
SMOVL C00316 +MOVJ EC00316
SMOVL C00317 +MOVJ EC00317
SMOVL C00318 +MOVJ EC00318
SMOVL C00319 +MOVJ EC00319
SMOVL C00320 +MOVJ EC00320
SMOVL C00321 +MOVJ EC00321
SMOVL C00322 +MOVJ EC00322
SMOVL C00323 +MOVJ EC00323
SMOVL C00324 +MOVJ EC00324
SMOVL C00325 +MOVJ EC00325
SMOVL C00326 +MOVJ EC00326
SMOVL C00327 +MOVJ EC00327
SMOVL C00328 +MOVJ EC00328
SMOVL C00329 +MOVJ EC00329
SMOVL C00330 +MOVJ EC00330
SMOVL C00331 +MOVJ EC00331
SMOVL C00332 +MOVJ EC00332
SMOVL C00333 +MOVJ EC00333
SMOVL C00334 +MOVJ EC00334
SMOVL C00335 +MOVJ EC00335
SMOVL C00336 +MOVJ EC00336
SMOVL C00337 +MOVJ EC00337
SMOVL C00338 +MOVJ EC00338
SMOVL C00339 +MOVJ EC00339
SMOVL C00340 +MOVJ EC00340
SMOVL C00341 +MOVJ EC00341
SMOVL C00342 +MOVJ EC00342
SMOVL C00343 +MOVJ EC00343
SMOVL C00344 +MOVJ EC00344
SMOVL C00345 +MOVJ EC00345
SMOVL C00346 +MOVJ EC00346
SMOVL C00347 +MOVJ EC00347
SMOVL C00348 +MOVJ EC00348
SMOVL C00349 +MOVJ EC00349
SMOVL C00350 +MOVJ EC00350
SMOVL C00351 +MOVJ EC00351
SMOVL C00352 +MOVJ EC00352
SMOVL C00353 +MOVJ EC00353
SMOVL C00354 +MOVJ EC00354
SMOVL C00355 +MOVJ EC00355
SMOVL C00356 +MOVJ EC00356
SMOVL C00357 +MOVJ EC00357
SMOVL C00358 +MOVJ EC00358
SMOVL C00359 +MOVJ EC00359
SMOVL C00360 +MOVJ EC00360
SMOVL C00361 +MOVJ EC00361
SMOVL C00362 +MOVJ EC00362
SMOVL C00363 +MOVJ EC00363
SMOVL C00364 +MOVJ EC00364
SMOVL C00365 +MOVJ EC00365
SMOVL C00366 +MOVJ EC00366
SMOVL C00367 +MOVJ EC00367
SMOVL C00368 +MOVJ EC00368
SMOVL C00369 +MOVJ EC00369
SMOVL C00370 +MOVJ EC00370
SMOVL C00371 +MOVJ EC00371
SMOVL C00372 +MOVJ EC00372
SMOVL C00373 +MOVJ EC00373
SMOVL C00374 +MOVJ EC00374
SMOVL C00375 +MOVJ EC00375
SMOVL C00376 +MOVJ EC00376
SMOVL C00377 +MOVJ EC00377
SMOVL C00378 +MOVJ EC00378
SMOVL C00379 +MOVJ EC00379
SMOVL C00380 +MOVJ EC00380
SMOVL C00381 +MOVJ EC00381
SMOVL C00382 +MOVJ EC00382
SMOVL C00383 +MOVJ EC00383
SMOVL C00384 +MOVJ EC00384
SMOVL C00385 +MOVJ EC00385
SMOVL C00386 +MOVJ EC00386
SMOVL C00387 +MOVJ EC00387
SMOVL C00388 +MOVJ EC00388
SMOVL C00389 +MOVJ EC00389
SMOVL C00390 +MOVJ EC00390
SMOVL C00391 +MOVJ EC00391
SMOVL C00392 +MOVJ EC00392
SMOVL C00393 +MOVJ EC00393
SMOVL C00394 +MOVJ EC00394
SMOVL C00395 +MOVJ EC00395
SMOVL C00396 +MOVJ EC00396
SMOVL C00397 +MOVJ EC00397
SMOVL C00398 +MOVJ EC00398
SMOVL C00399 +MOVJ EC00399
SMOVL C00400 +MOVJ EC00400
SMOVL C00401 +MOVJ EC00401
SMOVL C00402 +MOVJ EC00402
SMOVL C00403 +MOVJ EC00403
SMOVL C00404 +MOVJ EC00404
SMOVL C00405 +MOVJ EC00405
SMOVL C00406 +MOVJ EC00406
SMOVL C00407 +MOVJ EC00407
SMOVL C00408 +MOVJ EC00408
SMOVL C00409 +MOVJ EC00409
SMOVL C00410 +MOVJ EC00410
SMOVL C00411 +MOVJ EC00411
SMOVL C00412 +MOVJ EC00412
SMOVL C00413 +MOVJ EC00413
SMOVL C00414 +MOVJ EC00414
SMOVL C00415 +MOVJ EC00415
SMOVL C00416 +MOVJ EC00416
SMOVL C00417 +MOVJ EC00417
SMOVL C00418 +MOVJ EC00418
SMOVL C00419 +MOVJ EC00419
SMOVL C00420 +MOVJ EC00420
SMOVL C00421 +MOVJ EC00421
SMOVL C00422 +MOVJ EC00422
SMOVL C00423 +MOVJ EC00423
SMOVL C00424 +MOVJ EC00424
SMOVL C00425 +MOVJ EC00425
SMOVL C00426 +MOVJ EC00426
SMOVL C00427 +MOVJ EC00427
SMOVL C00428 +MOVJ EC00428
SMOVL C00429 +MOVJ EC00429
SMOVL C00430 +MOVJ EC00430
SMOVL C00431 +MOVJ EC00431
SMOVL C00432 +MOVJ EC00432
SMOVL C00433 +MOVJ EC00433
SMOVL C00434 +MOVJ EC00434
SMOVL C00435 +MOVJ EC00435
SMOVL C00436 +MOVJ EC00436
SMOVL C00437 +MOVJ EC00437
SMOVL C00438 +MOVJ EC00438
SMOVL C00439 +MOVJ EC00439
SMOVL C00440 +MOVJ EC00440
SMOVL C00441 +MOVJ EC00441
SMOVL C00442 +MOVJ EC00442
SMOVL C00443 +MOVJ EC00443
SMOVL C00444 +MOVJ EC00444
SMOVL C00445 +MOVJ EC00445
SMOVL C00446 +MOVJ EC00446
SMOVL C00447 +MOVJ EC00447
SMOVL C00448 +MOVJ EC00448
SMOVL C00449 +MOVJ EC00449
SMOVL C00450 +MOVJ EC00450
SMOVL C00451 +MOVJ EC00451
SMOVL C00452 +MOVJ EC00452
SMOVL C00453 +MOVJ EC00453
SMOVL C00454 +MOVJ EC00454
SMOVL C00455 +MOVJ EC00455
SMOVL C00456 +MOVJ EC00456
SMOVL C00457 +MOVJ EC00457
SMOVL C00458 +MOVJ EC00458
SMOVL C00459 +MOVJ EC00459
SMOVL C00460 +MOVJ EC00460
SMOVL C00461 +MOVJ EC00461
SMOVL C00462 +MOVJ EC00462
SMOVL C00463 +MOVJ EC00463
SMOVL C00464 +MOVJ EC00464
SMOVL C00465 +MOVJ EC00465
SMOVL C00466 +MOVJ EC00466
SMOVL C00467 +MOVJ EC00467
SMOVL C00468 +MOVJ EC00468
SMOVL C00469 +MOVJ EC00469
SMOVL C00470 +MOVJ EC00470
SMOVL C00471 +MOVJ EC00471
SMOVL C00472 +MOVJ EC00472
SMOVL C00473 +MOVJ EC00473
SMOVL C00474 +MOVJ EC00474
SMOVL C00475 +MOVJ EC00475
SMOVL C00476 +MOVJ EC00476
SMOVL C00477 +MOVJ EC00477
SMOVL C00478 +MOVJ EC00478
SMOVL C00479 +MOVJ EC00479
SMOVL C00480 +MOVJ EC00480
SMOVL C00481 +MOVJ EC00481
SMOVL C00482 +MOVJ EC00482
SMOVL C00483 +MOVJ EC00483
SMOVL C00484 +MOVJ EC00484
SMOVL C00485 +MOVJ EC00485
SMOVL C00486 +MOVJ EC00486
SMOVL C00487 +MOVJ EC00487
SMOVL C00488 +MOVJ EC00488
SMOVL C00489 +MOVJ EC00489
SMOVL C00490 +MOVJ EC00490
SMOVL C00491 +MOVJ EC00491
SMOVL C00492 +MOVJ EC00492
SMOVL C00493 +MOVJ EC00493
SMOVL C00494 +MOVJ EC00494
SMOVL C00495 +MOVJ EC00495
SMOVL C00496 +MOVJ EC00496
SMOVL C00497 +MOVJ EC00497
SMOVL C00498 +MOVJ EC00498
SMOVL C00499 +MOVJ EC00499
SMOVL C00500 +MOVJ EC00500
SMOVL C00501 +MOVJ EC00501
SMOVL C00502 +MOVJ EC00502
SMOVL C00503 +MOVJ EC00503
SMOVL C00504 +MOVJ EC00504
SMOVL C00505 +MOVJ EC00505
SMOVL C00506 +MOVJ EC00506
SMOVL C00507 +MOVJ EC00507
SMOVL C00508 +MOVJ EC00508
SMOVL C00509 +MOVJ EC00509
SMOVL C00510 +MOVJ EC00510
SMOVL C00511 +MOVJ EC00511
SMOVL C00512 +MOVJ EC00512
SMOVL C00513 +MOVJ EC00513
SMOVL C00514 +MOVJ EC00514
SMOVL C00515 +MOVJ EC00515
SMOVL C00516 +MOVJ EC00516
SMOVL C00517 +MOVJ EC00517
SMOVL C00518 +MOVJ EC00518
SMOVL C00519 +MOVJ EC00519
SMOVL C00520 +MOVJ EC00520
SMOVL C00521 +MOVJ EC00521
SMOVL C00522 +MOVJ EC00522
SMOVL C00523 +MOVJ EC00523
SMOVL C00524 +MOVJ EC00524
SMOVL C00525 +MOVJ EC00525
SMOVL C00526 +MOVJ EC00526
SMOVL C00527 +MOVJ EC00527
SMOVL C00528 +MOVJ EC00528
SMOVL C00529 +MOVJ EC00529
SMOVL C00530 +MOVJ EC00530
SMOVL C00531 +MOVJ EC00531
SMOVL C00532 +MOVJ EC00532
SMOVL C00533 +MOVJ EC00533
SMOVL C00534 +MOVJ EC00534
SMOVL C00535 +MOVJ EC00535
SMOVL C00536 +MOVJ EC00536
SMOVL C00537 +MOVJ EC00537
SMOVL C00538 +MOVJ EC00538
SMOVL C00539 +MOVJ EC00539
SMOVL C00540 +MOVJ EC00540
SMOVL C00541 +MOVJ EC00541
SMOVL C00542 +MOVJ EC00542
SMOVL C00543 +MOVJ EC00543
SMOVL C00544 +MOVJ EC00544
SMOVL C00545 +MOVJ EC00545
SMOVL C00546 +MOVJ EC00546
SMOVL C00547 +MOVJ EC00547
SMOVL C00548 +MOVJ EC00548
SMOVL C00549 +MOVJ EC00549
SMOVL C00550 +MOVJ EC00550
SMOVL C00551 +MOVJ EC00551
SMOVL C00552 +MOVJ EC00552
SMOVL C00553 +MOVJ EC00553
SMOVL C00554 +MOVJ EC00554
SMOVL C00555 +MOVJ EC00555
SMOVL C00556 +MOVJ EC00556
SMOVL C00557 +MOVJ EC00557
SMOVL C00558 +MOVJ EC00558
SMOVL C00559 +MOVJ EC00559
SMOVL C00560 +MOVJ EC00560
SMOVL C00561 +MOVJ EC00561
SMOVL C00562 +MOVJ EC00562
SMOVL C00563 +MOVJ EC00563
SMOVL C00564 +MOVJ EC00564
SMOVL C00565 +MOVJ EC00565
SMOVL C00566 +MOVJ EC00566
SMOVL C00567 +MOVJ EC00567
SMOVL C00568 +MOVJ EC00568
SMOVL C00569 +MOVJ EC00569
SMOVL C00570 +MOVJ EC00570
SMOVL C00571 +MOVJ EC00571
SMOVL C00572 +MOVJ EC00572
SMOVL C00573 +MOVJ EC00573
SMOVL C00574 +MOVJ EC00574
SMOVL C00575 +MOVJ EC00575
SMOVL C00576 +MOVJ EC00576
SMOVL C00577 +MOVJ EC00577
SMOVL C00578 +MOVJ EC00578
SMOVL C00579 +MOVJ EC00579
SMOVL C00580 +MOVJ EC00580
SMOVL C00581 +MOVJ EC00581
SMOVL C00582 +MOVJ EC00582
SMOVL C00583 +MOVJ EC00583
SMOVL C00584 +MOVJ EC00584
SMOVL C00585 +MOVJ EC00585
SMOVL C00586 +MOVJ EC00586
SMOVL C00587 +MOVJ EC00587
SMOVL C00588 +MOVJ EC00588
SMOVL C00589 +MOVJ EC00589
SMOVL C00590 +MOVJ EC00590
SMOVL C00591 +MOVJ EC00591
SMOVL C00592 +MOVJ EC00592
SMOVL C00593 +MOVJ EC00593
SMOVL C00594 +MOVJ EC00594
SMOVL C00595 +MOVJ EC00595
SMOVL C00596 +MOVJ EC00596
SMOVL C00597 +MOVJ EC00597
SMOVL C00598 +MOVJ EC00598
SMOVL C00599 +MOVJ EC00599
SMOVL C00600 +MOVJ EC00600
SMOVL C00601 +MOVJ EC00601
SMOVL C00602 +MOVJ EC00602
SMOVL C00603 +MOVJ EC00603
SMOVL C00604 +MOVJ EC00604
SMOVL C00605 +MOVJ EC00605
SMOVL C00606 +MOVJ EC00606
SMOVL C00607 +MOVJ EC00607
SMOVL C00608 +MOVJ EC00608
SMOVL C00609 +MOVJ EC00609
SMOVL C00610 +MOVJ EC00610
SMOVL C00611 +MOVJ EC00611
SMOVL C00612 +MOVJ EC00612
SMOVL C00613 +MOVJ EC00613
SMOVL C00614 +MOVJ EC00614
SMOVL C00615 +MOVJ EC00615
SMOVL C00616 +MOVJ EC00616
SMOVL C00617 +MOVJ EC00617
SMOVL C00618 +MOVJ EC00618
SMOVL C00619 +MOVJ EC00619
SMOVL C00620 +MOVJ EC00620
SMOVL C00621 +MOVJ EC00621
SMOVL C00622 +MOVJ EC00622
SMOVL C00623 +MOVJ EC00623
SMOVL C00624 +MOVJ EC00624
SMOVL C00625 +MOVJ EC00625
SMOVL C00626 +MOVJ EC00626
SMOVL C00627 +MOVJ EC00627
SMOVL C00628 +MOVJ EC00628
SMOVL C00629 +MOVJ EC00629
SMOVL C00630 +MOVJ EC00630
SMOVL C00631 +MOVJ EC00631
SMOVL C00632 +MOVJ EC00632
SMOVL C00633 +MOVJ EC00633
SMOVL C00634 +MOVJ EC00634
SMOVL C00635 +MOVJ EC00635
SMOVL C00636 +MOVJ EC00636
SMOVL C00637 +MOVJ EC00637
SMOVL C00638 +MOVJ EC00638
SMOVL C00639 +MOVJ EC00639
SMOVL C00640 +MOVJ EC00640
SMOVL C00641 +MOVJ EC00641
SMOVL C00642 +MOVJ EC00642
SMOVL C00643 +MOVJ EC00643
SMOVL C00644 +MOVJ EC00644
SMOVL C00645 +MOVJ EC00645
SMOVL C00646 +MOVJ EC00646
SMOVL C00647 +MOVJ EC00647
SMOVL C00648 +MOVJ EC00648
SMOVL C00649 +MOVJ EC00649
SMOVL C00650 +MOVJ EC00650
SMOVL C00651 +MOVJ EC00651
SMOVL C00652 +MOVJ EC00652
SMOVL C00653 +MOVJ EC00653
SMOVL C00654 +MOVJ EC00654
SMOVL C00655 +MOVJ EC00655
SMOVL C00656 +MOVJ EC00656
SMOVL C00657 +MOVJ EC00657
SMOVL C00658 +MOVJ EC00658
SMOVL C00659 +MOVJ EC00659
SMOVL C00660 +MOVJ EC00660
SMOVL C00661 +MOVJ EC00661
SMOVL C00662 +MOVJ EC00662
SMOVL C00663 +MOVJ EC00663
SMOVL C00664 +MOVJ EC00664
SMOVL C00665 +MOVJ EC00665
SMOVL C00666 +MOVJ EC00666
SMOVL C00667 +MOVJ EC00667
SMOVL C00668 +MOVJ EC00668
SMOVL C00669 +MOVJ EC00669
SMOVL C00670 +MOVJ EC00670
SMOVL C00671 +MOVJ EC00671
SMOVL C00672 +MOVJ EC00672
SMOVL C00673 +MOVJ EC00673
SMOVL C00674 +MOVJ EC00674
SMOVL C00675 +MOVJ EC00675
SMOVL C00676 +MOVJ EC00676
SMOVL C00677 +MOVJ EC00677
SMOVL C00678 +MOVJ EC00678
SMOVL C00679 +MOVJ EC00679
SMOVL C00680 +MOVJ EC00680
SMOVL C00681 +MOVJ EC00681
SMOVL C00682 +MOVJ EC00682
SMOVL C00683 +MOVJ EC00683
SMOVL C00684 +MOVJ EC00684
SMOVL C00685 +MOVJ EC00685
SMOVL C00686 +MOVJ EC00686
SMOVL C00687 +MOVJ EC00687
SMOVL C00688 +MOVJ EC00688
SMOVL C00689 +MOVJ EC00689
SMOVL C00690 +MOVJ EC00690
SMOVL C00691 +MOVJ EC00691
SMOVL C00692 +MOVJ EC00692
SMOVL C00693 +MOVJ EC00693
SMOVL C00694 +MOVJ EC00694
SMOVL C00695 +MOVJ EC00695
SMOVL C00696 +MOVJ EC00696
SMOVL C00697 +MOVJ EC00697
SMOVL C00698 +MOVJ EC00698
SMOVL C00699 +MOVJ EC00699
SMOVL C00700 +MOVJ EC00700
SMOVL C00701 +MOVJ EC00701
SMOVL C00702 +MOVJ EC00702
SMOVL C00703 +MOVJ EC00703
SMOVL C00704 +MOVJ EC00704
SMOVL C00705 +MOVJ EC00705
SMOVL C00706 +MOVJ EC00706
SMOVL C00707 +MOVJ EC00707
SMOVL C00708 +MOVJ EC00708
SMOVL C00709 +MOVJ EC00709
SMOVL C00710 +MOVJ EC00710
SMOVL C00711 +MOVJ EC00711
SMOVL C00712 +MOVJ EC00712
SMOVL C00713 +MOVJ EC00713
SMOVL C00714 +MOVJ EC00714
SMOVL C00715 +MOVJ EC00715
SMOVL C00716 +MOVJ EC00716
SMOVL C00717 +MOVJ EC00717
SMOVL C00718 +MOVJ EC00718
SMOVL C00719 +MOVJ EC00719
SMOVL C00720 +MOVJ EC00720
SMOVL C00721 +MOVJ EC00721
SMOVL C00722 +MOVJ EC00722
SMOVL C00723 +MOVJ EC00723
SMOVL C00724 +MOVJ EC00724
SMOVL C00725 +MOVJ EC00725
SMOVL C00726 +MOVJ EC00726
SMOVL C00727 +MOVJ EC00727
SMOVL C00728 +MOVJ EC00728
SMOVL C00729 +MOVJ EC00729
SMOVL C00730 +MOVJ EC00730
SMOVL C00731 +MOVJ EC00731
SMOVL C00732 +MOVJ EC00732
SMOVL C00733 +MOVJ EC00733
SMOVL C00734 +MOVJ EC00734
SMOVL C00735 +MOVJ EC00735
SMOVL C00736 +MOVJ EC00736
SMOVL C00737 +MOVJ EC00737
SMOVL C00738 +MOVJ EC00738
SMOVL C00739 +MOVJ EC00739
SMOVL C00740 +MOVJ EC00740
SMOVL C00741 +MOVJ EC00741
SMOVL C00742 +MOVJ EC00742
SMOVL C00743 +MOVJ EC00743
SMOVL C00744 +MOVJ EC00744
SMOVL C00745 +MOVJ EC00745
SMOVL C00746 +MOVJ EC00746
SMOVL C00747 +MOVJ EC00747
SMOVL C00748 +MOVJ EC00748
SMOVL C00749 +MOVJ EC00749
SMOVL C00750 +MOVJ EC00750
SMOVL C00751 +MOVJ EC00751
SMOVL C00752 +MOVJ EC00752
SMOVL C00753 +MOVJ EC00753
SMOVL C00754 +MOVJ EC00754
SMOVL C00755 +MOVJ EC00755
SMOVL C00756 +MOVJ EC00756
SMOVL C00757 +MOVJ EC00757
SMOVL C00758 +MOVJ EC00758
SMOVL C00759 +MOVJ EC00759
SMOVL C00760 +MOVJ EC00760
SMOVL C00761 +MOVJ EC00761
SMOVL C00762 +MOVJ EC00762
SMOVL C00763 +MOVJ EC00763
SMOVL C00764 +MOVJ EC00764
SMOVL C00765 +MOVJ EC00765
SMOVL C00766 +MOVJ EC00766
SMOVL C00767 +MOVJ EC00767
SMOVL C00768 +MOVJ EC00768
SMOVL C00769 +MOVJ EC00769
SMOVL C00770 +MOVJ EC00770
SMOVL C00771 +MOVJ EC00771
SMOVL C00772 +MOVJ EC00772
SMOVL C00773 +MOVJ EC00773
SMOVL C00774 +MOVJ EC00774
SMOVL C00775 +MOVJ EC00775
SMOVL C00776 +MOVJ EC00776
SMOVL C00777 +MOVJ EC00777
SMOVL C00778 +MOVJ EC00778
SMOVL C00779 +MOVJ EC00779
SMOVL C00780 +MOVJ EC00780
SMOVL C00781 +MOVJ EC00781
SMOVL C00782 +MOVJ EC00782
SMOVL C00783 +MOVJ EC00783
SMOVL C00784 +MOVJ EC00784
SMOVL C00785 +MOVJ EC00785
SMOVL C00786 +MOVJ EC00786
SMOVL C00787 +MOVJ EC00787
SMOVL C00788 +MOVJ EC00788
SMOVL C00789 +MOVJ EC00789
SMOVL C00790 +MOVJ EC00790
SMOVL C00791 +MOVJ EC00791
SMOVL C00792 +MOVJ EC00792
SMOVL C00793 +MOVJ EC00793
SMOVL C00794 +MOVJ EC00794
SMOVL C00795 +MOVJ EC00795
SMOVL C00796 +MOVJ EC00796
SMOVL C00797 +MOVJ EC00797
SMOVL C00798 +MOVJ EC00798
SMOVL C00799 +MOVJ EC00799
SMOVL C00800 +MOVJ EC00800
SMOVL C00801 +MOVJ EC00801
SMOVL C00802 +MOVJ EC00802
SMOVL C00803 +MOVJ EC00803
SMOVL C00804 +MOVJ EC00804
SMOVL C00805 +MOVJ EC00805
SMOVL C00806 +MOVJ EC00806
SMOVL C00807 +MOVJ EC00807
SMOVL C00808 +MOVJ EC00808
SMOVL C00809 +MOVJ EC00809
SMOVL C00810 +MOVJ EC00810
SMOVL C00811 +MOVJ EC00811
SMOVL C00812 +MOVJ EC00812
SMOVL C00813 +MOVJ EC00813
SMOVL C00814 +MOVJ EC00814
SMOVL C00815 +MOVJ EC00815
SMOVL C00816 +MOVJ EC00816
SMOVL C00817 +MOVJ EC00817
SMOVL C00818 +MOVJ EC00818
SMOVL C00819 +MOVJ EC00819
SMOVL C00820 +MOVJ EC00820
SMOVL C00821 +MOVJ EC00821
SMOVL C00822 +MOVJ EC00822
SMOVL C00823 +MOVJ EC00823
SMOVL C00824 +MOVJ EC00824
SMOVL C00825 +MOVJ EC00825
SMOVL C00826 +MOVJ EC00826
SMOVL C00827 +MOVJ EC00827
SMOVL C00828 +MOVJ EC00828
SMOVL C00829 +MOVJ EC00829
SMOVL C00830 +MOVJ EC00830
SMOVL C00831 +MOVJ EC00831
SMOVL C00832 +MOVJ EC00832
SMOVL C00833 +MOVJ EC00833
SMOVL C00834 +MOVJ EC00834
SMOVL C00835 +MOVJ EC00835
SMOVL C00836 +MOVJ EC00836
SMOVL C00837 +MOVJ EC00837
SMOVL C00838 +MOVJ EC00838
SMOVL C00839 +MOVJ EC00839
SMOVL C00840 +MOVJ EC00840
SMOVL C00841 +MOVJ EC00841
SMOVL C00842 +MOVJ EC00842
SMOVL C00843 +MOVJ EC00843
SMOVL C00844 +MOVJ EC00844
SMOVL C00845 +MOVJ EC00845
SMOVL C00846 +MOVJ EC00846
SMOVL C00847 +MOVJ EC00847
SMOVL C00848 +MOVJ EC00848
SMOVL C00849 +MOVJ EC00849
SMOVL C00850 +MOVJ EC00850
SMOVL C00851 +MOVJ EC00851
SMOVL C00852 +MOVJ EC00852
SMOVL C00853 +MOVJ EC00853
SMOVL C00854 +MOVJ EC00854
SMOVL C00855 +MOVJ EC00855
SMOVL C00856 +MOVJ EC00856
SMOVL C00857 +MOVJ EC00857
SMOVL C00858 +MOVJ EC00858
SMOVL C00859 +MOVJ EC00859
SMOVL C00860 +MOVJ EC00860
SMOVL C00861 +MOVJ EC00861
SMOVL C00862 +MOVJ EC00862
SMOVL C00863 +MOVJ EC00863
SMOVL C00864 +MOVJ EC00864
SMOVL C00865 +MOVJ EC00865
SMOVL C00866 +MOVJ EC00866
SMOVL C00867 +MOVJ EC00867
SMOVL C00868 +MOVJ EC00868
SMOVL C00869 +MOVJ EC00869
SMOVL C00870 +MOVJ EC00870
SMOVL C00871 +MOVJ EC00871
SMOVL C00872 +MOVJ EC00872
SMOVL C00873 +MOVJ EC00873
SMOVL C00874 +MOVJ EC00874
SMOVL C00875 +MOVJ EC00875
SMOVL C00876 +MOVJ EC00876
SMOVL C00877 +MOVJ EC00877
SMOVL C00878 +MOVJ EC00878
SMOVL C00879 +MOVJ EC00879
SMOVL C00880 +MOVJ EC00880
SMOVL C00881 +MOVJ EC00881
SMOVL C00882 +MOVJ EC00882
SMOVL C00883 +MOVJ EC00883
SMOVL C00884 +MOVJ EC00884
SMOVL C00885 +MOVJ EC00885
SMOVL C00886 +MOVJ EC00886
SMOVL C00887 +MOVJ EC00887
SMOVL C00888 +MOVJ EC00888
SMOVL C00889 +MOVJ EC00889
SMOVL C00890 +MOVJ EC00890
SMOVL C00891 +MOVJ EC00891
SMOVL C00892 +MOVJ EC00892
SMOVL C00893 +MOVJ EC00893
SMOVL C00894 +MOVJ EC00894
SMOVL C00895 +MOVJ EC00895
SMOVL C00896 +MOVJ EC00896
SMOVL C00897 +MOVJ EC00897
SMOVL C00898 +MOVJ EC00898
SMOVL C00899 +MOVJ EC00899
SMOVL C00900 +MOVJ EC00900
SMOVL C00901 +MOVJ EC00901
SMOVL C00902 +MOVJ EC00902
SMOVL C00903 +MOVJ EC00903
SMOVL C00904 +MOVJ EC00904
SMOVL C00905 +MOVJ EC00905
SMOVL C00906 +MOVJ EC00906
SMOVL C00907 +MOVJ EC00907
SMOVL C00908 +MOVJ EC00908
SMOVL C00909 +MOVJ EC00909
SMOVL C00910 +MOVJ EC00910
SMOVL C00911 +MOVJ EC00911
SMOVL C00912 +MOVJ EC00912
SMOVL C00913 +MOVJ EC00913
SMOVL C00914 +MOVJ EC00914
SMOVL C00915 +MOVJ EC00915
SMOVL C00916 +MOVJ EC00916
SMOVL C00917 +MOVJ EC00917
SMOVL C00918 +MOVJ EC00918
SMOVL C00919 +MOVJ EC00919
SMOVL C00920 +MOVJ EC00920
SMOVL C00921 +MOVJ EC00921
SMOVL C00922 +MOVJ EC00922
SMOVL C00923 +MOVJ EC00923
SMOVL C00924 +MOVJ EC00924
SMOVL C00925 +MOVJ EC00925
SMOVL C00926 +MOVJ EC00926
SMOVL C00927 +MOVJ EC00927
SMOVL C00928 +MOVJ EC00928
SMOVL C00929 +MOVJ EC00929
SMOVL C00930 +MOVJ EC00930
SMOVL C00931 +MOVJ EC00931
SMOVL C00932 +MOVJ EC00932
SMOVL C00933 +MOVJ EC00933
SMOVL C00934 +MOVJ EC00934
SMOVL C00935 +MOVJ EC00935
SMOVL C00936 +MOVJ EC00936
SMOVL C00937 +MOVJ EC00937
SMOVL C00938 +MOVJ EC00938
SMOVL C00939 +MOVJ EC00939
SMOVL C00940 +MOVJ EC00940
SMOVL C00941 +MOVJ EC00941
SMOVL C00942 +MOVJ EC00942
SMOVL C00943 +MOVJ EC00943
SMOVL C00944 +MOVJ EC00944
SMOVL C00945 +MOVJ EC00945
SMOVL C00946 +MOVJ EC00946
SMOVL C00947 +MOVJ EC00947
SMOVL C00948 +MOVJ EC00948
SMOVL C00949 +MOVJ EC00949
SMOVL C00950 +MOVJ EC00950
SMOVL C00951 +MOVJ EC00951
SMOVL C00952 +MOVJ EC00952
SMOVL C00953 +MOVJ EC00953
SMOVL C00954 +MOVJ EC00954
SMOVL C00955 +MOVJ EC00955
SMOVL C00956 +MOVJ EC00956
SMOVL C00957 +MOVJ EC00957
SMOVL C00958 +MOVJ EC00958
SMOVL C00959 +MOVJ EC00959
SMOVL C00960 +MOVJ EC00960
SMOVL C00961 +MOVJ EC00961
SMOVL C00962 +MOVJ EC00962
SMOVL C00963 +MOVJ EC00963
SMOVL C00964 +MOVJ EC00964
SMOVL C00965 +MOVJ EC00965
SMOVL C00966 +MOVJ EC00966
SMOVL C00967 +MOVJ EC00967
SMOVL C00968 +MOVJ EC00968
SMOVL C00969 +MOVJ EC00969
SMOVL C00970 +MOVJ EC00970
SMOVL C00971 +MOVJ EC00971
SMOVL C00972 +MOVJ EC00972
SMOVL C00973 +MOVJ EC00973
SMOVL C00974 +MOVJ EC00974
SMOVL C00975 +MOVJ EC00975
SMOVL C00976 +MOVJ EC00976
SMOVL C00977 +MOVJ EC00977
SMOVL C00978 +MOVJ EC00978
SMOVL C00979 +MOVJ EC00979
SMOVL C00980 +MOVJ EC00980
SMOVL C00981 +MOVJ EC00981
SMOVL C00982 +MOVJ EC00982
SMOVL C00983 +MOVJ EC00983
SMOVL C00984 +MOVJ EC00984
SMOVL C00985 +MOVJ EC00985
SMOVL C00986 +MOVJ EC00986
SMOVL C00987 +MOVJ EC00987
SMOVL C00988 +MOVJ EC00988
SMOVL C00989 +MOVJ EC00989
SMOVL C00990 +MOVJ EC00990
SMOVL C00991 +MOVJ EC00991
SMOVL C00992 +MOVJ EC00992
SMOVL C00993 +MOVJ EC00993
SMOVL C00994 +MOVJ EC00994
SMOVL C00995 +MOVJ EC00995
SMOVL C00996 +MOVJ EC00996
SMOVL C00997 +MOVJ EC00997
SMOVL C00998 +MOVJ EC00998
SMOVL C00999 +MOVJ EC00999
SMOVL C01000 +MOVJ EC01000
SMOVL C01001 +MOVJ EC01001
SMOVL C01002 +MOVJ EC01002
SMOVL C01003 +MOVJ EC01003
SMOVL C01004 +MOVJ EC01004
SMOVL C01005 +MOVJ EC01005
SMOVL C01006 +MOVJ EC01006
SMOVL C01007 +MOVJ EC01007
SMOVL C01008 +MOVJ EC01008
SMOVL C01009 +MOVJ EC01009
SMOVL C01010 +MOVJ EC01010
SMOVL C01011 +MOVJ EC01011
SMOVL C01012 +MOVJ EC01012
SMOVL C01013 +MOVJ EC01013
SMOVL C01014 +MOVJ EC01014
SMOVL C01015 +MOVJ EC01015
SMOVL C01016 +MOVJ EC01016
SMOVL C01017 +MOVJ EC01017
SMOVL C01018 +MOVJ EC01018
SMOVL C01019 +MOVJ EC01019
SMOVL C01020 +MOVJ EC01020
SMOVL C01021 +MOVJ EC01021
SMOVL C01022 +MOVJ EC01022
SMOVL C01023 +MOVJ EC01023
SMOVL C01024 +MOVJ EC01024
SMOVL C01025 +MOVJ EC01025
SMOVL C01026 +MOVJ EC01026
SMOVL C01027 +MOVJ EC01027
SMOVL C01028 +MOVJ EC01028
SMOVL C01029 +MOVJ EC01029
SMOVL C01030 +MOVJ EC01030
SMOVL C01031 +MOVJ EC01031
SMOVL C01032 +MOVJ EC01032
SMOVL C01033 +MOVJ EC01033
SMOVL C01034 +MOVJ EC01034
SMOVL C01035 +MOVJ EC01035
SMOVL C01036 +MOVJ EC01036
SMOVL C01037 +MOVJ EC01037
SMOVL C01038 +MOVJ EC01038
SMOVL C01039 +MOVJ EC01039
SMOVL C01040 +MOVJ EC01040
SMOVL C01041 +MOVJ EC01041
SMOVL C01042 +MOVJ EC01042
SMOVL C01043 +MOVJ EC01043
SMOVL C01044 +MOVJ EC01044
SMOVL C01045 +MOVJ EC01045
SMOVL C01046 +MOVJ EC01046
SMOVL C01047 +MOVJ EC01047
SMOVL C01048 +MOVJ EC01048
SMOVL C01049 +MOVJ EC01049
SMOVL C01050 +MOVJ EC01050
SMOVL C01051 +MOVJ EC01051
SMOVL C01052 +MOVJ EC01052
SMOVL C01053 +MOVJ EC01053
SMOVL C01054 +MOVJ EC01054
SMOVL C01055 +MOVJ EC01055
SMOVL C01056 +MOVJ EC01056
SMOVL C01057 +MOVJ EC01057
SMOVL C01058 +MOVJ EC01058
SMOVL C01059 +MOVJ EC01059
SMOVL C01060 +MOVJ EC01060
SMOVL C01061 +MOVJ EC01061
SMOVL C01062 +MOVJ EC01062
SMOVL C01063 +MOVJ EC01063
SMOVL C01064 +MOVJ EC01064
SMOVL C01065 +MOVJ EC01065
SMOVL C01066 +MOVJ EC01066
SMOVL C01067 +MOVJ EC01067
SMOVL C01068 +MOVJ EC01068
SMOVL C01069 +MOVJ EC01069
SMOVL C01070 +MOVJ EC01070
SMOVL C01071 +MOVJ EC01071
SMOVL C01072 +MOVJ EC01072
SMOVL C01073 +MOVJ EC01073
SMOVL C01074 +MOVJ EC01074
SMOVL C01075 +MOVJ EC01075
SMOVL C01076 +MOVJ EC01076
SMOVL C01077 +MOVJ EC01077
SMOVL C01078 +MOVJ EC01078
SMOVL C01079 +MOVJ EC01079
SMOVL C01080 +MOVJ EC01080
SMOVL C01081 +MOVJ EC01081
SMOVL C01082 +MOVJ EC01082
SMOVL C01083 +MOVJ EC01083
SMOVL C01084 +MOVJ EC01084
SMOVL C01085 +MOVJ EC01085
SMOVL C01086 +MOVJ EC01086
SMOVL C01087 +MOVJ EC01087
SMOVL C01088 +MOVJ EC01088
SMOVL C01089 +MOVJ EC01089
SMOVL C01090 +MOVJ EC01090
SMOVL C01091 +MOVJ EC01091
SMOVL C01092 +MOVJ EC01092
SMOVL C01093 +MOVJ EC01093
SMOVL C01094 +MOVJ EC01094
SMOVL C01095 +MOVJ EC01095
SMOVL C01096 +MOVJ EC01096
SMOVL C01097 +MOVJ EC01097
SMOVL C01098 +MOVJ EC01098
SMOVL C01099 +MOVJ EC01099
SMOVL C01100 +MOVJ EC01100
SMOVL C01101 +MOVJ EC01101
SMOVL C01102 +MOVJ EC01102
SMOVL C01103 +MOVJ EC01103
SMOVL C01104 +MOVJ EC01104
SMOVL C01105 +MOVJ EC01105
SMOVL C01106 +MOVJ EC01106
SMOVL C01107 +MOVJ EC01107
SMOVL C01108 +MOVJ EC01108
SMOVL C01109 +MOVJ EC01109
SMOVL C01110 +MOVJ EC01110
SMOVL C01111 +MOVJ EC01111
SMOVL C01112 +MOVJ EC01112
SMOVL C01113 +MOVJ EC01113
SMOVL C01114 +MOVJ EC01114
SMOVL C01115 +MOVJ EC01115
SMOVL C01116 +MOVJ EC01116
SMOVL C01117 +MOVJ EC01117
SMOVL C01118 +MOVJ EC01118
SMOVL C01119 +MOVJ EC01119
SMOVL C01120 +MOVJ EC01120
SMOVL C01121 +MOVJ EC01121
SMOVL C01122 +MOVJ EC01122
SMOVL C01123 +MOVJ EC01123
SMOVL C01124 +MOVJ EC01124
SMOVL C01125 +MOVJ EC01125
SMOVL C01126 +MOVJ EC01126
SMOVL C01127 +MOVJ EC01127
SMOVL C01128 +MOVJ EC01128
SMOVL C01129 +MOVJ EC01129
SMOVL C01130 +MOVJ EC01130
SMOVL C01131 +MOVJ EC01131
SMOVL C01132 +MOVJ EC01132
SMOVL C01133 +MOVJ EC01133
SMOVL C01134 +MOVJ EC01134
SMOVL C01135 +MOVJ EC01135
SMOVL C01136 +MOVJ EC01136
SMOVL C01137 +MOVJ EC01137
SMOVL C01138 +MOVJ EC01138
SMOVL C01139 +MOVJ EC01139
SMOVL C01140 +MOVJ EC01140
SMOVL C01141 +MOVJ EC01141
SMOVL C01142 +MOVJ EC01142
SMOVL C01143 +MOVJ EC01143
SMOVL C01144 +MOVJ EC01144
SMOVL C01145 +MOVJ EC01145
SMOVL C01146 +MOVJ EC01146
SMOVL C01147 +MOVJ EC01147
SMOVL C01148 +MOVJ EC01148
SMOVL C01149 +MOVJ EC01149
SMOVL C01150 +MOVJ EC01150
SMOVL C01151 +MOVJ EC01151
SMOVL C01152 +MOVJ EC01152
SMOVL C01153 +MOVJ EC01153
SMOVL C01154 +MOVJ EC01154
SMOVL C01155 +MOVJ EC01155
SMOVL C01156 +MOVJ EC01156
SMOVL C01157 +MOVJ EC01157
SMOVL C01158 +MOVJ EC01158
SMOVL C01159 +MOVJ EC01159
SMOVL C01160 +MOVJ EC01160
SMOVL C01161 +MOVJ EC01161
SMOVL C01162 +MOVJ EC01162
SMOVL C01163 +MOVJ EC01163
SMOVL C01164 +MOVJ EC01164
SMOVL C01165 +MOVJ EC01165
SMOVL C01166 +MOVJ EC01166
SMOVL C01167 +MOVJ EC01167
SMOVL C01168 +MOVJ EC01168
SMOVL C01169 +MOVJ EC01169
SMOVL C01170 +MOVJ EC01170
SMOVL C01171 +MOVJ EC01171
SMOVL C01172 +MOVJ EC01172
SMOVL C01173 +MOVJ EC01173
SMOVL C01174 +MOVJ EC01174
SMOVL C01175 +MOVJ EC01175
SMOVL C01176 +MOVJ EC01176
SMOVL C01177 +MOVJ EC01177
SMOVL C01178 +MOVJ EC01178
SMOVL C01179 +MOVJ EC01179
SMOVL C01180 +MOVJ EC01180
SMOVL C01181 +MOVJ EC01181
SMOVL C01182 +MOVJ EC01182
SMOVL C01183 +MOVJ EC01183
SMOVL C01184 +MOVJ EC01184
SMOVL C01185 +MOVJ EC01185
SMOVL C01186 +MOVJ EC01186
SMOVL C01187 +MOVJ EC01187
SMOVL C01188 +MOVJ EC01188
SMOVL C01189 +MOVJ EC01189
SMOVL C01190 +MOVJ EC01190
SMOVL C01191 +MOVJ EC01191
SMOVL C01192 +MOVJ EC01192
SMOVL C01193 +MOVJ EC01193
SMOVL C01194 +MOVJ EC01194
SMOVL C01195 +MOVJ EC01195
SMOVL C01196 +MOVJ EC01196
SMOVL C01197 +MOVJ EC01197
SMOVL C01198 +MOVJ EC01198
SMOVL C01199 +MOVJ EC01199
SMOVL C01200 +MOVJ EC01200
SMOVL C01201 +MOVJ EC01201
SMOVL C01202 +MOVJ EC01202
SMOVL C01203 +MOVJ EC01203
SMOVL C01204 +MOVJ EC01204
SMOVL C01205 +MOVJ EC01205
SMOVL C01206 +MOVJ EC01206
SMOVL C01207 +MOVJ EC01207
SMOVL C01208 +MOVJ EC01208
SMOVL C01209 +MOVJ EC01209
SMOVL C01210 +MOVJ EC01210
SMOVL C01211 +MOVJ EC01211
SMOVL C01212 +MOVJ EC01212
SMOVL C01213 +MOVJ EC01213
SMOVL C01214 +MOVJ EC01214
SMOVL C01215 +MOVJ EC01215
SMOVL C01216 +MOVJ EC01216
SMOVL C01217 +MOVJ EC01217
SMOVL C01218 +MOVJ EC01218
SMOVL C01219 +MOVJ EC01219
SMOVL C01220 +MOVJ EC01220
SMOVL C01221 +MOVJ EC01221
SMOVL C01222 +MOVJ EC01222
SMOVL C01223 +MOVJ EC01223
SMOVL C01224 +MOVJ EC01224
SMOVL C01225 +MOVJ EC01225
SMOVL C01226 +MOVJ EC01226
SMOVL C01227 +MOVJ EC01227
SMOVL C01228 +MOVJ EC01228
SMOVL C01229 +MOVJ EC01229
SMOVL C01230 +MOVJ EC01230
SMOVL C01231 +MOVJ EC01231
SMOVL C01232 +MOVJ EC01232
SMOVL C01233 +MOVJ EC01233
SMOVL C01234 +MOVJ EC01234
SMOVL C01235 +MOVJ EC01235
SMOVL C01236 +MOVJ EC01236
SMOVL C01237 +MOVJ EC01237
SMOVL C01238 +MOVJ EC01238
SMOVL C01239 +MOVJ EC01239
SMOVL C01240 +MOVJ EC01240
SMOVL C01241 +MOVJ EC01241
SMOVL C01242 +MOVJ EC01242
SMOVL C01243 +MOVJ EC01243
SMOVL C01244 +MOVJ EC01244
SMOVL C01245 +MOVJ EC01245
SMOVL C01246 +MOVJ EC01246
SMOVL C01247 +MOVJ EC01247
SMOVL C01248 +MOVJ EC01248
SMOVL C01249 +MOVJ EC01249
SMOVL C01250 +MOVJ EC01250
SMOVL C01251 +MOVJ EC01251
SMOVL C01252 +MOVJ EC01252
SMOVL C01253 +MOVJ EC01253
SMOVL C01254 +MOVJ EC01254
SMOVL C01255 +MOVJ EC01255
SMOVL C01256 +MOVJ EC01256
SMOVL C01257 +MOVJ EC01257
SMOVL C01258 +MOVJ EC01258
SMOVL C01259 +MOVJ EC01259
SMOVL C01260 +MOVJ EC01260
SMOVL C01261 +MOVJ EC01261
SMOVL C01262 +MOVJ EC01262
SMOVL C01263 +MOVJ EC01263
SMOVL C01264 +MOVJ EC01264
SMOVL C01265 +MOVJ EC01265
SMOVL C01266 +MOVJ EC01266
SMOVL C01267 +MOVJ EC01267
SMOVL C01268 +MOVJ EC01268
SMOVL C01269 +MOVJ EC01269
SMOVL C01270 +MOVJ EC01270
SMOVL C01271 +MOVJ EC01271
SMOVL C01272 +MOVJ EC01272
SMOVL C01273 +MOVJ EC01273
SMOVL C01274 +MOVJ EC01274
SMOVL C01275 +MOVJ EC01275
SMOVL C01276 +MOVJ EC01276
SMOVL C01277 +MOVJ EC01277
SMOVL C01278 +MOVJ EC01278
SMOVL C01279 +MOVJ EC01279
SMOVL C01280 +MOVJ EC01280
SMOVL C01281 +MOVJ EC01281
SMOVL C01282 +MOVJ EC01282
SMOVL C01283 +MOVJ EC01283
SMOVL C01284 +MOVJ EC01284
SMOVL C01285 +MOVJ EC01285
SMOVL C01286 +MOVJ EC01286
SMOVL C01287 +MOVJ EC01287
SMOVL C01288 +MOVJ EC01288
SMOVL C01289 +MOVJ EC01289
SMOVL C01290 +MOVJ EC01290
SMOVL C01291 +MOVJ EC01291
SMOVL C01292 +MOVJ EC01292
SMOVL C01293 +MOVJ EC01293
SMOVL C01294 +MOVJ EC01294
SMOVL C01295 +MOVJ EC01295
SMOVL C01296 +MOVJ EC01296
SMOVL C01297 +MOVJ EC01297
SMOVL C01298 +MOVJ EC01298
SMOVL C01299 +MOVJ EC01299
SMOVL C01300 +MOVJ EC01300
SMOVL C01301 +MOVJ EC01301
SMOVL C01302 +MOVJ EC01302
SMOVL C01303 +MOVJ EC01303
SMOVL C01304 +MOVJ EC01304
SMOVL C01305 +MOVJ EC01305
SMOVL C01306 +MOVJ EC01306
SMOVL C01307 +MOVJ EC01307
SMOVL C01308 +MOVJ EC01308
SMOVL C01309 +MOVJ EC01309
SMOVL C01310 +MOVJ EC01310
SMOVL C01311 +MOVJ EC01311
SMOVL C01312 +MOVJ EC01312
SMOVL C01313 +MOVJ EC01313
SMOVL C01314 +MOVJ EC01314
SMOVL C01315 +MOVJ EC01315
SMOVL C01316 +MOVJ EC01316
SMOVL C01317 +MOVJ EC01317
SMOVL C01318 +MOVJ EC01318
SMOVL C01319 +MOVJ EC01319
SMOVL C01320 +MOVJ EC01320
SMOVL C01321 +MOVJ EC01321
SMOVL C01322 +MOVJ EC01322
SMOVL C01323 +MOVJ EC01323
SMOVL C01324 +MOVJ EC01324
SMOVL C01325 +MOVJ EC01325
SMOVL C01326 +MOVJ EC01326
SMOVL C01327 +MOVJ EC01327
SMOVL C01328 +MOVJ EC01328
SMOVL C01329 +MOVJ EC01329
SMOVL C01330 +MOVJ EC01330
SMOVL C01331 +MOVJ EC01331
SMOVL C01332 +MOVJ EC01332
SMOVL C01333 +MOVJ EC01333
SMOVL C01334 +MOVJ EC01334
SMOVL C01335 +MOVJ EC01335
SMOVL C01336 +MOVJ EC01336
SMOVL C01337 +MOVJ EC01337
SMOVL C01338 +MOVJ EC01338
SMOVL C01339 +MOVJ EC01339
SMOVL C01340 +MOVJ EC01340
SMOVL C01341 +MOVJ EC01341
SMOVL C01342 +MOVJ EC01342
SMOVL C01343 +MOVJ EC01343
SMOVL C01344 +MOVJ EC01344
SMOVL C01345 +MOVJ EC01345
SMOVL C01346 +MOVJ EC01346
SMOVL C01347 +MOVJ EC01347
SMOVL C01348 +MOVJ EC01348
SMOVL C01349 +MOVJ EC01349
SMOVL C01350 +MOVJ EC01350
SMOVL C01351 +MOVJ EC01351
SMOVL C01352 +MOVJ EC01352
SMOVL C01353 +MOVJ EC01353
SMOVL C01354 +MOVJ EC01354
SMOVL C01355 +MOVJ EC01355
SMOVL C01356 +MOVJ EC01356
SMOVL C01357 +MOVJ EC01357
SMOVL C01358 +MOVJ EC01358
SMOVL C01359 +MOVJ EC01359
SMOVL C01360 +MOVJ EC01360
SMOVL C01361 +MOVJ EC01361
SMOVL C01362 +MOVJ EC01362
SMOVL C01363 +MOVJ EC01363
SMOVL C01364 +MOVJ EC01364
SMOVL C01365 +MOVJ EC01365
SMOVL C01366 +MOVJ EC01366
SMOVL C01367 +MOVJ EC01367
SMOVL C01368 +MOVJ EC01368
SMOVL C01369 +MOVJ EC01369
SMOVL C01370 +MOVJ EC01370
SMOVL C01371 +MOVJ EC01371
SMOVL C01372 +MOVJ EC01372
SMOVL C01373 +MOVJ EC01373
SMOVL C01374 +MOVJ EC01374
SMOVL C01375 +MOVJ EC01375
SMOVL C01376 +MOVJ EC01376
SMOVL C01377 +MOVJ EC01377
SMOVL C01378 +MOVJ EC01378
SMOVL C01379 +MOVJ EC01379
SMOVL C01380 +MOVJ EC01380
SMOVL C01381 +MOVJ EC01381
SMOVL C01382 +MOVJ EC01382
SMOVL C01383 +MOVJ EC01383
SMOVL C01384 +MOVJ EC01384
SMOVL C01385 +MOVJ EC01385
SMOVL C01386 +MOVJ EC01386
SMOVL C01387 +MOVJ EC01387
SMOVL C01388 +MOVJ EC01388
SMOVL C01389 +MOVJ EC01389
SMOVL C01390 +MOVJ EC01390
SMOVL C01391 +MOVJ EC01391
SMOVL C01392 +MOVJ EC01392
SMOVL C01393 +MOVJ EC01393
SMOVL C01394 +MOVJ EC01394
SMOVL C01395 +MOVJ EC01395
SMOVL C01396 +MOVJ EC01396
SMOVL C01397 +MOVJ EC01397
SMOVL C01398 +MOVJ EC01398
SMOVL C01399 +MOVJ EC01399
SMOVL C01400 +MOVJ EC01400
SMOVL C01401 +MOVJ EC01401
SMOVL C01402 +MOVJ EC01402
SMOVL C01403 +MOVJ EC01403
SMOVL C01404 +MOVJ EC01404
SMOVL C01405 +MOVJ EC01405
SMOVL C01406 +MOVJ EC01406
SMOVL C01407 +MOVJ EC01407
SMOVL C01408 +MOVJ EC01408
SMOVL C01409 +MOVJ EC01409
SMOVL C01410 +MOVJ EC01410
SMOVL C01411 +MOVJ EC01411
SMOVL C01412 +MOVJ EC01412
SMOVL C01413 +MOVJ EC01413
SMOVL C01414 +MOVJ EC01414
SMOVL C01415 +MOVJ EC01415
SMOVL C01416 +MOVJ EC01416
SMOVL C01417 +MOVJ EC01417
SMOVL C01418 +MOVJ EC01418
SMOVL C01419 +MOVJ EC01419
SMOVL C01420 +MOVJ EC01420
SMOVL C01421 +MOVJ EC01421
SMOVL C01422 +MOVJ EC01422
SMOVL C01423 +MOVJ EC01423
SMOVL C01424 +MOVJ EC01424
SMOVL C01425 +MOVJ EC01425
SMOVL C01426 +MOVJ EC01426
SMOVL C01427 +MOVJ EC01427
SMOVL C01428 +MOVJ EC01428
SMOVL C01429 +MOVJ EC01429
SMOVL C01430 +MOVJ EC01430
SMOVL C01431 +MOVJ EC01431
SMOVL C01432 +MOVJ EC01432
SMOVL C01433 +MOVJ EC01433
SMOVL C01434 +MOVJ EC01434
SMOVL C01435 +MOVJ EC01435
SMOVL C01436 +MOVJ EC01436
SMOVL C01437 +MOVJ EC01437
SMOVL C01438 +MOVJ EC01438
SMOVL C01439 +MOVJ EC01439
SMOVL C01440 +MOVJ EC01440
SMOVL C01441 +MOVJ EC01441
SMOVL C01442 +MOVJ EC01442
SMOVL C01443 +MOVJ EC01443
SMOVL C01444 +MOVJ EC01444
SMOVL C01445 +MOVJ EC01445
SMOVL C01446 +MOVJ EC01446
SMOVL C01447 +MOVJ EC01447
SMOVL C01448 +MOVJ EC01448
SMOVL C01449 +MOVJ EC01449
SMOVL C01450 +MOVJ EC01450
SMOVL C01451 +MOVJ EC01451
SMOVL C01452 +MOVJ EC01452
SMOVL C01453 +MOVJ EC01453
SMOVL C01454 +MOVJ EC01454
SMOVL C01455 +MOVJ EC01455
SMOVL C01456 +MOVJ EC01456
SMOVL C01457 +MOVJ EC01457
SMOVL C01458 +MOVJ EC01458
SMOVL C01459 +MOVJ EC01459
SMOVL C01460 +MOVJ EC01460
SMOVL C01461 +MOVJ EC01461
SMOVL C01462 +MOVJ EC01462
SMOVL C01463 +MOVJ EC01463
SMOVL C01464 +MOVJ EC01464
SMOVL C01465 +MOVJ EC01465
SMOVL C01466 +MOVJ EC01466
SMOVL C01467 +MOVJ EC01467
SMOVL C01468 +MOVJ EC01468
SMOVL C01469 +MOVJ EC01469
SMOVL C01470 +MOVJ EC01470
SMOVL C01471 +MOVJ EC01471
SMOVL C01472 +MOVJ EC01472
SMOVL C01473 +MOVJ EC01473
SMOVL C01474 +MOVJ EC01474
SMOVL C01475 +MOVJ EC01475
SMOVL C01476 +MOVJ EC01476
SMOVL C01477 +MOVJ EC01477
SMOVL C01478 +MOVJ EC01478
SMOVL C01479 +MOVJ EC01479
SMOVL C01480 +MOVJ EC01480
SMOVL C01481 +MOVJ EC01481
SMOVL C01482 +MOVJ EC01482
SMOVL C01483 +MOVJ EC01483
SMOVL C01484 +MOVJ EC01484
SMOVL C01485 +MOVJ EC01485
SMOVL C01486 +MOVJ EC01486
SMOVL C01487 +MOVJ EC01487
SMOVL C01488 +MOVJ EC01488
SMOVL C01489 +MOVJ EC01489
SMOVL C01490 +MOVJ EC01490
SMOVL C01491 +MOVJ EC01491
SMOVL C01492 +MOVJ EC01492
SMOVL C01493 +MOVJ EC01493
SMOVL C01494 +MOVJ EC01494
SMOVL C01495 +MOVJ EC01495
SMOVL C01496 +MOVJ EC01496
SMOVL C01497 +MOVJ EC01497
SMOVL C01498 +MOVJ EC01498
SMOVL C01499 +MOVJ EC01499
SMOVL C01500 +MOVJ EC01500
SMOVL C01501 +MOVJ EC01501
SMOVL C01502 +MOVJ EC01502
SMOVL C01503 +MOVJ EC01503
SMOVL C01504 +MOVJ EC01504
SMOVL C01505 +MOVJ EC01505
SMOVL C01506 +MOVJ EC01506
SMOVL C01507 +MOVJ EC01507
SMOVL C01508 +MOVJ EC01508
SMOVL C01509 +MOVJ EC01509
SMOVL C01510 +MOVJ EC01510
SMOVL C01511 +MOVJ EC01511
SMOVL C01512 +MOVJ EC01512
SMOVL C01513 +MOVJ EC01513
SMOVL C01514 +MOVJ EC01514
SMOVL C01515 +MOVJ EC01515
SMOVL C01516 +MOVJ EC01516
SMOVL C01517 +MOVJ EC01517
SMOVL C01518 +MOVJ EC01518
SMOVL C01519 +MOVJ EC01519
SMOVL C01520 +MOVJ EC01520
SMOVL C01521 +MOVJ EC01521
SMOVL C01522 +MOVJ EC01522
SMOVL C01523 +MOVJ EC01523
SMOVL C01524 +MOVJ EC01524
SMOVL C01525 +MOVJ EC01525
SMOVL C01526 +MOVJ EC01526
SMOVL C01527 +MOVJ EC01527
SMOVL C01528 +MOVJ EC01528
SMOVL C01529 +MOVJ EC01529
SMOVL C01530 +MOVJ EC01530
SMOVL C01531 +MOVJ EC01531
SMOVL C01532 +MOVJ EC01532
SMOVL C01533 +MOVJ EC01533
SMOVL C01534 +MOVJ EC01534
SMOVL C01535 +MOVJ EC01535
SMOVL C01536 +MOVJ EC01536
SMOVL C01537 +MOVJ EC01537
SMOVL C01538 +MOVJ EC01538
SMOVL C01539 +MOVJ EC01539
SMOVL C01540 +MOVJ EC01540
SMOVL C01541 +MOVJ EC01541
SMOVL C01542 +MOVJ EC01542
SMOVL C01543 +MOVJ EC01543
SMOVL C01544 +MOVJ EC01544
SMOVL C01545 +MOVJ EC01545
SMOVL C01546 +MOVJ EC01546
SMOVL C01547 +MOVJ EC01547
SMOVL C01548 +MOVJ EC01548
SMOVL C01549 +MOVJ EC01549
SMOVL C01550 +MOVJ EC01550
SMOVL C01551 +MOVJ EC01551
SMOVL C01552 +MOVJ EC01552
SMOVL C01553 +MOVJ EC01553
SMOVL C01554 +MOVJ EC01554
SMOVL C01555 +MOVJ EC01555
SMOVL C01556 +MOVJ EC01556
SMOVL C01557 +MOVJ EC01557
SMOVL C01558 +MOVJ EC01558
SMOVL C01559 +MOVJ EC01559
SMOVL C01560 +MOVJ EC01560
SMOVL C01561 +MOVJ EC01561
SMOVL C01562 +MOVJ EC01562
SMOVL C01563 +MOVJ EC01563
SMOVL C01564 +MOVJ EC01564
SMOVL C01565 +MOVJ EC01565
SMOVL C01566 +MOVJ EC01566
SMOVL C01567 +MOVJ EC01567
SMOVL C01568 +MOVJ EC01568
SMOVL C01569 +MOVJ EC01569
SMOVL C01570 +MOVJ EC01570
SMOVL C01571 +MOVJ EC01571
SMOVL C01572 +MOVJ EC01572
SMOVL C01573 +MOVJ EC01573
SMOVL C01574 +MOVJ EC01574
SMOVL C01575 +MOVJ EC01575
SMOVL C01576 +MOVJ EC01576
SMOVL C01577 +MOVJ EC01577
SMOVL C01578 +MOVJ EC01578
SMOVL C01579 +MOVJ EC01579
SMOVL C01580 +MOVJ EC01580
SMOVL C01581 +MOVJ EC01581
SMOVL C01582 +MOVJ EC01582
SMOVL C01583 +MOVJ EC01583
SMOVL C01584 +MOVJ EC01584
SMOVL C01585 +MOVJ EC01585
SMOVL C01586 +MOVJ EC01586
SMOVL C01587 +MOVJ EC01587
SMOVL C01588 +MOVJ EC01588
SMOVL C01589 +MOVJ EC01589
SMOVL C01590 +MOVJ EC01590
SMOVL C01591 +MOVJ EC01591
SMOVL C01592 +MOVJ EC01592
SMOVL C01593 +MOVJ EC01593
SMOVL C01594 +MOVJ EC01594
SMOVL C01595 +MOVJ EC01595
SMOVL C01596 +MOVJ EC01596
SMOVL C01597 +MOVJ EC01597
SMOVL C01598 +MOVJ EC01598
SMOVL C01599 +MOVJ EC01599
SMOVL C01600 +MOVJ EC01600
SMOVL C01601 +MOVJ EC01601
SMOVL C01602 +MOVJ EC01602
SMOVL C01603 +MOVJ EC01603
SMOVL C01604 +MOVJ EC01604
SMOVL C01605 +MOVJ EC01605
SMOVL C01606 +MOVJ EC01606
SMOVL C01607 +MOVJ EC01607
SMOVL C01608 +MOVJ EC01608
SMOVL C01609 +MOVJ EC01609
SMOVL C01610 +MOVJ EC01610
SMOVL C01611 +MOVJ EC01611
SMOVL C01612 +MOVJ EC01612
SMOVL C01613 +MOVJ EC01613
SMOVL C01614 +MOVJ EC01614
SMOVL C01615 +MOVJ EC01615
SMOVL C01616 +MOVJ EC01616
SMOVL C01617 +MOVJ EC01617
SMOVL C01618 +MOVJ EC01618
SMOVL C01619 +MOVJ EC01619
SMOVL C01620 +MOVJ EC01620
SMOVL C01621 +MOVJ EC01621
SMOVL C01622 +MOVJ EC01622
SMOVL C01623 +MOVJ EC01623
SMOVL C01624 +MOVJ EC01624
SMOVL C01625 +MOVJ EC01625
SMOVL C01626 +MOVJ EC01626
SMOVL C01627 +MOVJ EC01627
SMOVL C01628 +MOVJ EC01628
SMOVL C01629 +MOVJ EC01629
SMOVL C01630 +MOVJ EC01630
SMOVL C01631 +MOVJ EC01631
SMOVL C01632 +MOVJ EC01632
SMOVL C01633 +MOVJ EC01633
SMOVL C01634 +MOVJ EC01634
SMOVL C01635 +MOVJ EC01635
SMOVL C01636 +MOVJ EC01636
SMOVL C01637 +MOVJ EC01637
SMOVL C01638 +MOVJ EC01638
SMOVL C01639 +MOVJ EC01639
SMOVL C01640 +MOVJ EC01640
SMOVL C01641 +MOVJ EC01641
SMOVL C01642 +MOVJ EC01642
SMOVL C01643 +MOVJ EC01643
SMOVL C01644 +MOVJ EC01644
SMOVL C01645 +MOVJ EC01645
SMOVL C01646 +MOVJ EC01646
SMOVL C01647 +MOVJ EC01647
SMOVL C01648 +MOVJ EC01648
SMOVL C01649 +MOVJ EC01649
SMOVL C01650 +MOVJ EC01650
SMOVL C01651 +MOVJ EC01651
SMOVL C01652 +MOVJ EC01652
SMOVL C01653 +MOVJ EC01653
SMOVL C01654 +MOVJ EC01654
SMOVL C01655 +MOVJ EC01655
SMOVL C01656 +MOVJ EC01656
SMOVL C01657 +MOVJ EC01657
SMOVL C01658 +MOVJ EC01658
SMOVL C01659 +MOVJ EC01659
SMOVL C01660 +MOVJ EC01660
SMOVL C01661 +MOVJ EC01661
SMOVL C01662 +MOVJ EC01662
SMOVL C01663 +MOVJ EC01663
SMOVL C01664 +MOVJ EC01664
SMOVL C01665 +MOVJ EC01665
SMOVL C01666 +MOVJ EC01666
SMOVL C01667 +MOVJ EC01667
SMOVL C01668 +MOVJ EC01668
SMOVL C01669 +MOVJ EC01669
SMOVL C01670 +MOVJ EC01670
SMOVL C01671 +MOVJ EC01671
SMOVL C01672 +MOVJ EC01672
SMOVL C01673 +MOVJ EC01673
SMOVL C01674 +MOVJ EC01674
SMOVL C01675 +MOVJ EC01675
SMOVL C01676 +MOVJ EC01676
SMOVL C01677 +MOVJ EC01677
SMOVL C01678 +MOVJ EC01678
SMOVL C01679 +MOVJ EC01679
SMOVL C01680 +MOVJ EC01680
SMOVL C01681 +MOVJ EC01681
SMOVL C01682 +MOVJ EC01682
SMOVL C01683 +MOVJ EC01683
SMOVL C01684 +MOVJ EC01684
